    if(wv_seq[0] == 0 or wv_seq[0] == 3):
      if(a9_wv_weldingon==True):
        program_weld_on = False
        if(isHicomm):
          write_port_register(202,0)
          write_port_register(149,0)
        else:
          set_standard_digital_out(0,False)
        end
        if(wv_weldpar[2]==1):
          target_pos = feature_offset(get_actual_tcp_pose(),p[0,0,-0.01,0,0,0],wv_Line_Feature2)
          movel(target_pos,0.5,0.01)
        end
      end
    end
    background_pose = [dumy_p,dumy_p,dumy_p,dumy_p]
    move_p = background_pose
    return sin_dir
  end
  $ 151 "Reset"
  $ 152 "If Reset_Trig"
  if (Reset_Trig):
    $ 153 "Reset_Trig≔ False "
    global Reset_Trig=  False
    $ 154 "Call robotand_cell_initalizat"
    robotand_cell_initalizat()
    $ 155 "Auto_trig≔ False "
    global Auto_trig=  False
    $ 156 "write_port_register(cell_3f_2f_151,0)"
    write_port_register(cell_3f_2f_151,0)
    $ 157 "write_port_register(cell_info_152,0)"
    write_port_register(cell_info_152,0)
    $ 158 "write_port_register(weld_req_153,0)"
    write_port_register(weld_req_153,0)
    $ 159 "write_port_register(return_done_240,0)"
    write_port_register(return_done_240,0)
    $ 160 "write_port_register(robot_move_163,0)"
    write_port_register(robot_move_163,0)
    $ 161 "write_port_register(robot_pose_164,0)"
    write_port_register(robot_pose_164,0)
    $ 162 "write_port_register(182,0)"
    write_port_register(182,0)
    $ 163 "write_port_register(185,0)"
    write_port_register(185,0)
    $ 164 "write_port_register(201,0)"
    write_port_register(201,0)
    $ 165 "write_port_register(202,0)"
    write_port_register(202,0)
  end
  $ 166 "Welding_Init"
  $ 167 "'welding parameter initialization'"
  # 'welding parameter initialization'
  $ 168 "welding_etc"
  $ 196 "c5_wv_gap_y≔0"
  global c5_wv_gap_y=0
  $ 197 "c6_wv_gap_cpm≔0"
  global c6_wv_gap_cpm=0
  $ 198 "c9_wv_gap_freq≔0"
  global c9_wv_gap_freq=0
  $ 199 "c4_gap_enable≔0"
  global c4_gap_enable=0
  $ 200 "c7_wv_gap≔[c4_gap_enable,c5_wv_gap_y,c6_wv_gap_cpm,c9_wv_gap_freq]"
  global c7_wv_gap=[c4_gap_enable,c5_wv_gap_y,c6_wv_gap_cpm,c9_wv_gap_freq]
  $ 201 "init_reset_modbus_server"
  $ 202 "set_tool_voltage(24)"
  set_tool_voltage(24)
  $ 203 "write_port_register(163,0)"
  write_port_register(163,0)
  $ 204 "write_port_register(164,0)"
  write_port_register(164,0)
  $ 206 "write_port_register(201,1)"
  write_port_register(201,1)
  $ 207 "write_port_register(202,0)"
  write_port_register(202,0)
  $ 1277 "Thread_2"
  thread Thread_2():
    while (True):
      $ 1278 "Thread_heartbeat"
      $ 1279 "heartbeat≔heartbeat+1"
      global heartbeat=heartbeat+1
      $ 1280 "If heartbeat>499"
      if (heartbeat>499):
        $ 1281 "heartbeat≔0"
        global heartbeat=0
      end
      $ 1282 "write_port_register(128,heartbeat)"
      write_port_register(128,heartbeat)
      $ 1292 "Wait: 1.0"
      sleep(1.0)
    end
  end
  threadId_Thread_2 = run Thread_2()
  $ 1293 "Thread_1"
  thread Thread_1():
    while (True):
      $ 1294 "thread main"
      $ 1295 "a0_Job_Mode≔read_port_register(162)"
      global a0_Job_Mode= read_port_register (162)
      $ 1296 "a1_job_move≔read_port_register(163)"
      global a1_job_move= read_port_register (163)
      $ 1297 "If red_led≟ True "
      if (get_tool_digital_out(0) ==   True  ):
        $ 1298 "Set red_led=Off"
        set_tool_digital_out(0, False)
      end
      $ 1299 "If a0_Job_Mode≟2"
      if (a0_Job_Mode == 2):
        $ 1300 "If read_port_register(arc_onoff_168)≟2"
        if ( read_port_register (arc_onoff_168) == 2):
          $ 1301 "a9_wv_weldingon≔ True "
          global a9_wv_weldingon=  True
        else:
          $ 1302 "Else" "noBreak"
          $ 1303 "a9_wv_weldingon≔ False "
          global a9_wv_weldingon=  False
        end
        $ 1304 "If Auto_trig"
        if (Auto_trig):
          $ 1305 "get_next_number≔read_port_register(166)"
          global get_next_number= read_port_register (166)
          $ 1306 "get_move_trig≔read_port_register(167)"
          global get_move_trig= read_port_register (167)
          $ 1307 "If get_move_trig≟1 and running_trig≟ True "
          if (get_move_trig == 1  and  running_trig ==   True  ):
            $ 1308 "If get_next_number<0 or get_next_number>30"
            if (get_next_number<0  or  get_next_number>30):
              $ 1309 "write_port_register(142,141)"
              write_port_register(142,141)
              $ 1310 "Halt"
              halt
            end
            $ 1311 "If get_next_number≠Auto_cur_cell"
            if (get_next_number != Auto_cur_cell):
              $ 1312 "running_trig≔ False "
              global running_trig=  False
              $ 1313 "write_welder(0, False )"
              write_welder(0,  False  )
              $ 1314 "write_port_register(149,0)"
              write_port_register(149,0)
              $ 1315 "write_port_register(202,0)"
              write_port_register(202,0)
            else:
              $ 1316 "Else" "noBreak"
              $ 1317 "write_port_register(166,0)"
              write_port_register(166,0)
              $ 1318 "write_port_register(167,0)"
              write_port_register(167,0)
            end
          end
        end
        $ 1319 "If t_time>timer_1"
        if (t_time>timer_1):
          $ 1320 "write_port_register(143,timer_1)"
          write_port_register(143,timer_1)
        else:
          $ 1321 "Else" "noBreak"
          $ 1322 "write_port_register(143,timer_1)"
          write_port_register(143,timer_1)
          $ 1323 "write_port_register(144,timer_1)"
          write_port_register(144,timer_1)
        end
        $ 1324 "Monitoring touch and welding"
        $ 1325 "If read_welder_control(0) and read_port_register(130)≠1"
        if (read_welder_control(0)  and   read_port_register (130) != 1):
          $ 1326 "write_port_register(130,1)"
          write_port_register(130,1)
        else:
          $ 1327 "ElseIf read_welder_control(0) and read_port_register(130)≠0"
          if (read_welder_control(0)  and   read_port_register (130) != 0):
            $ 1328 "write_port_register(130,0)"
            write_port_register(130,0)
          end
        end
        $ 1329 "If read_welder(5)"
        if (read_welder(5)):
          $ 1330 "'check wcr in (digital)'"
          # 'check wcr in (digital)'
          $ 1331 "write_output_float_register(20,1)"
          write_output_float_register(20,1)
        else:
          $ 1332 "Else" "noBreak"
          $ 1333 "write_output_float_register(20,0)"
          write_output_float_register(20,0)
        end
        $ 1334 "If read_welder(4)"
        if (read_welder(4)):
          $ 1335 "'check touch (digital)'"
          # 'check touch (digital)'
          $ 1336 "write_output_float_register(21,1)"
          write_output_float_register(21,1)
        else:
          $ 1337 "Else" "noBreak"
          $ 1338 "write_output_float_register(21,0)"
          write_output_float_register(21,0)
        end
        $ 1339 "If read_welder_control(0)"
        if (read_welder_control(0)):
          $ 1340 "'check welding out (digital)'"
          # 'check welding out (digital)'
          $ 1341 "write_output_float_register(17,1)"
          write_output_float_register(17,1)
        else:
          $ 1342 "Else" "noBreak"
          $ 1343 "write_output_float_register(17,0)"
          write_output_float_register(17,0)
        end
        $ 1344 "If read_welder_control(4)"
        if (read_welder_control(4)):
          $ 1345 "'check touch out (digital)'"
          # 'check touch out (digital)'
          $ 1346 "write_output_float_register(18,1)"
          write_output_float_register(18,1)
        else:
          $ 1347 "Else" "noBreak"
          $ 1348 "write_output_float_register(18,0)"
          write_output_float_register(18,0)
        end
      end
      $ 1349 "If get_tool_digital_in(1)≟ True "
      if (get_tool_digital_in(1) ==   True  ):
        $ 1350 "set_tool_digital_out(1, False )"
        set_tool_digital_out(1,  False  )
      else:
        $ 1351 "Else" "noBreak"
        $ 1352 "set_tool_digital_out(1, True )"
        set_tool_digital_out(1,  True  )
      end
      $ 1353 "If red_led≟ True "
      if (get_tool_digital_out(0) ==   True  ):
        $ 1354 "Set red_led=Off"
        set_tool_digital_out(0, False)
        $ 1355 "end_freedrive_mode()"
        end_freedrive_mode()
      end
      $ 1356 "check_speed()"
      check_speed()
      $ 1357 "Wait: 0.05"
      sleep(0.05)
    end
  end
  threadId_Thread_1 = run Thread_1()
  thread EventThread():
    while (True):
      if (event_cal_on):
        $ 1359 "calculate_position"
        $ 1362 "move_i_f≔1"
        global move_i_f=1
        $ 1363 "get_pose_side≔0"
        global get_pose_side=0
        $ 1364 "Loop move_i_f<10"
        while (move_i_f<10):
          $ 1365 "If A_Touch_trig_l[move_i_f]≟ True "
          if (A_Touch_trig_l[move_i_f] ==   True  ):
            $ 1366 "If move_i_f≟A_VL1 or move_i_f≟A_VL2"
            if (move_i_f == A_VL1  or  move_i_f == A_VL2):
              $ 1367 "A_sel_v≔move_i_f"
              global A_sel_v=move_i_f
              $ 1368 "If simulation_mode"
              if (simulation_mode):
                $ 1369 "Call welding_parameter_sim"
                welding_parameter_sim()
              else:
                $ 1370 "Else" "noBreak"
                $ 1371 "Call welding_parameter_init"
                welding_parameter_init()
              end
              $ 1372 "If a8_wv_distance<5"
              if (a8_wv_distance<5):
                $ 1373 "write_port_register(142,143)"
                write_port_register(142,143)
                $ 1374 "Halt"
                halt
              end
              $ 1375 "b2_left_par≔ True "
              global b2_left_par=  True
              $ 1376 "b8_wv_2f≔ False "
              global b8_wv_2f=  False
              $ 1377 "If move_i_f≟A_VL2"
              if (move_i_f == A_VL2):
                $ 1378 "callar_hor≔a6_callar_hor"
                global callar_hor=a6_callar_hor
                $ 1379 "If b1_cell_info_L≟E or b1_cell_info_L≟e"
                if (b1_cell_info_L == E  or  b1_cell_info_L == e):
                  $ 1380 "'For bottom touch(zero) after offset not used now'"
                  # 'For bottom touch(zero) after offset not used now'
                  $ 1381 "vert_scallup_l≔a5_f_hole[1]"
                  global vert_scallup_l=a5_f_hole[1]
                end
                $ 1382 "b2_cell≔b1_cell_info_L"
                global b2_cell=b1_cell_info_L
              else:
                $ 1385 "Else" "noBreak"
                $ 1386 "callar_hor≔0"
                global callar_hor=0
                $ 1387 "'For bottom touch(zero) after offset not used now'"
                # 'For bottom touch(zero) after offset not used now'
                $ 1388 "vert_scallup_l≔a5_f_hole[1]"
                global vert_scallup_l=a5_f_hole[1]
                $ 1389 "b2_cell≔b1_cell_info_L"
                global b2_cell=b1_cell_info_L
              end
              $ 1390 "get_pos≔get_lr(left,a6_f_width,a5_f_hole,a7_f_distance,b2_left_par,b8_wv_2f,Touch_dis,get_margin_z,get_pose_side,callar_hor,b2_cell,center_line)"
              global get_pos=get_lr(p[.480496318984, .411279115151, .006998291210, -2.211681476386, -.899147924387, -1.383032568605],a6_f_width,a5_f_hole,a7_f_distance,b2_left_par,b8_wv_2f,Touch_dis,get_margin_z,get_pose_side,callar_hor,b2_cell,center_line)
              $ 1391 "pre_tp≔tilt_3f_fun(get_pos,[0,0,0],0)"
              global pre_tp=tilt_3f_fun(get_pos,[0,0,0],0)
              $ 1392 "A_Prepos_l[move_i_f]=pre_tp"
              A_Prepos_l[move_i_f]=pre_tp
            else:
              $ 1393 "ElseIf move_i_f≟A_VR1 or move_i_f≟A_VR2"
              if (move_i_f == A_VR1  or  move_i_f == A_VR2):
                $ 1394 "A_sel_v≔move_i_f"
                global A_sel_v=move_i_f
                $ 1395 "If simulation_mode"
                if (simulation_mode):
                  $ 1396 "Call welding_parameter_sim"
                  welding_parameter_sim()
                else:
                  $ 1397 "Else" "noBreak"
                  $ 1398 "Call welding_parameter_init"
                  welding_parameter_init()
                end
                $ 1399 "If a8_wv_distance<5"
                if (a8_wv_distance<5):
                  $ 1400 "write_port_register(142,143)"
                  write_port_register(142,143)
                  $ 1401 "Halt"
                  halt
                end
                $ 1402 "b2_left_par≔ False "
                global b2_left_par=  False
                $ 1403 "b8_wv_2f≔ False "
                global b8_wv_2f=  False
                $ 1404 "If move_i_f≟A_VR2"
                if (move_i_f == A_VR2):
                  $ 1405 "callar_hor≔a6_callar_hor"
                  global callar_hor=a6_callar_hor
                  $ 1406 "If b1_cell_info_R≟E or b1_cell_info_R≟e"
                  if (b1_cell_info_R == E  or  b1_cell_info_R == e):
                    $ 1407 "vert_scallup_r≔a5_f_hole[1]"
                    global vert_scallup_r=a5_f_hole[1]
                  end
                  $ 1408 "b2_cell≔b1_cell_info_R"
                  global b2_cell=b1_cell_info_R
                else:
                  $ 1411 "Else" "noBreak"
                  $ 1412 "callar_hor≔0"
                  global callar_hor=0
                  $ 1413 "vert_scallup_r≔a5_f_hole[1]"
                  global vert_scallup_r=a5_f_hole[1]
                  $ 1414 "b2_cell≔b1_cell_info_R"
                  global b2_cell=b1_cell_info_R
                end
                $ 1415 "get_pos≔get_lr(right,a6_f_width,a5_f_hole,a7_f_distance,b2_left_par,b8_wv_2f,Touch_dis,get_margin_z,get_pose_side,callar_hor,b2_cell,center_line)"
                global get_pos=get_lr(p[.475000000000, -.421403215678, .026417194146, 1.917761036827, -1.141682393512, 1.523356199292],a6_f_width,a5_f_hole,a7_f_distance,b2_left_par,b8_wv_2f,Touch_dis,get_margin_z,get_pose_side,callar_hor,b2_cell,center_line)
                $ 1416 "pre_tp≔tilt_3f_fun(get_pos,[0,0,0],0)"
                global pre_tp=tilt_3f_fun(get_pos,[0,0,0],0)
                $ 1417 "A_Prepos_l[move_i_f]=pre_tp"
                A_Prepos_l[move_i_f]=pre_tp
              else:
                $ 1418 "ElseIf move_i_f≟A_HOR"
                if (move_i_f == A_HOR):
                  $ 1419 "A_sel_v≔A_HOR"
                  global A_sel_v=A_HOR
                  $ 1420 "If simulation_mode"
                  if (simulation_mode):
                    $ 1421 "Call welding_parameter_sim"
                    welding_parameter_sim()
                  else:
                    $ 1422 "Else" "noBreak"
                    $ 1423 "Call welding_parameter_init"
                    welding_parameter_init()
                  end
                  $ 1424 "hor_l_scallup≔a5_f_hole[1]"
                  global hor_l_scallup=a5_f_hole[1]
                  $ 1425 "b8_wv_2f≔ True "
                  global b8_wv_2f=  True
                  $ 1426 "b2_left_par≔ True "
                  global b2_left_par=  True
                  $ 1427 "b2_cell≔b1_cell_info_L"
                  global b2_cell=b1_cell_info_L
                  $ 1428 "get_pos≔get_lr(up_left,a6_f_width,a5_f_hole,a7_f_distance,b2_left_par,b8_wv_2f,Touch_dis,get_margin_z,get_pose_side,0,b2_cell,center_line)"
                  global get_pos=get_lr(p[.492775857339, .409517380626, -.029063830209, -2.419264859926, -.998084331190, -1.368689080860],a6_f_width,a5_f_hole,a7_f_distance,b2_left_par,b8_wv_2f,Touch_dis,get_margin_z,get_pose_side,0,b2_cell,center_line)
                  $ 1429 "pre_tp≔get_pos"
                  global pre_tp=get_pos
                  $ 1430 "A_Prepos_l[move_i_f]=pre_tp"
                  A_Prepos_l[move_i_f]=pre_tp
                else:
                  $ 1431 "ElseIf move_i_f≟A_HOR_R"
                  if (move_i_f == A_HOR_R):
                    $ 1432 "A_sel_v≔A_HOR"
                    global A_sel_v=A_HOR
                    $ 1433 "If simulation_mode"
                    if (simulation_mode):
                      $ 1434 "Call welding_parameter_sim"
                      welding_parameter_sim()
                    else:
                      $ 1435 "Else" "noBreak"
                      $ 1436 "Call welding_parameter_init"
                      welding_parameter_init()
                    end
                    $ 1437 "hor_r_scallup≔a5_f_hole[2]"
                    global hor_r_scallup=a5_f_hole[2]
                    $ 1438 "b2_left_par≔ False "
                    global b2_left_par=  False
                    $ 1439 "b8_wv_2f≔ True "
                    global b8_wv_2f=  True
                    $ 1440 "b2_cell≔b1_cell_info_R"
                    global b2_cell=b1_cell_info_R
                    $ 1441 "get_pos≔get_lr(up_right,a6_f_width,a5_f_hole,a7_f_distance,b2_left_par,b8_wv_2f,Touch_dis,get_margin_z,get_pose_side,0,b2_cell,center_line)"
                    global get_pos=get_lr(p[.445203173045, -.406687378356, -.031125942276, 2.308490741423, -1.066468937023, 1.322151316133],a6_f_width,a5_f_hole,a7_f_distance,b2_left_par,b8_wv_2f,Touch_dis,get_margin_z,get_pose_side,0,b2_cell,center_line)
                    $ 1442 "pre_tp≔get_pos"
                    global pre_tp=get_pos
                    $ 1443 "A_Prepos_l[move_i_f]=pre_tp"
                    A_Prepos_l[move_i_f]=pre_tp
                  else:
                    $ 1444 "ElseIf move_i_f≟A_HOR_ML"
                    if (move_i_f == A_HOR_ML):
                      $ 1445 "A_sel_v≔A_HOR_ML"
                      global A_sel_v=A_HOR_ML
                      $ 1446 "If simulation_mode"
                      if (simulation_mode):
                        $ 1447 "Call welding_parameter_sim"
                        welding_parameter_sim()
                      else:
                        $ 1448 "Else" "noBreak"
                        $ 1449 "Call welding_parameter_init"
                        welding_parameter_init()
                      end
                      $ 1450 "b8_wv_2f≔ True "
                      global b8_wv_2f=  True
                      $ 1451 "b2_left_par≔ True "
                      global b2_left_par=  True
                      $ 1452 "b2_cell≔b1_cell_info_L"
                      global b2_cell=b1_cell_info_L
                      $ 1453 "Touch_dis≔-1*Touch_dis"
                      global Touch_dis=-1*Touch_dis
                      $ 1454 "get_pos≔get_lr(up_left,a6_f_width,a5_f_hole,a7_f_distance,b2_left_par,b8_wv_2f,Touch_dis,get_margin_z,get_pose_side,a6_callar_hor,b2_cell,center_line)"
                      global get_pos=get_lr(p[.492775857339, .409517380626, -.029063830209, -2.419264859926, -.998084331190, -1.368689080860],a6_f_width,a5_f_hole,a7_f_distance,b2_left_par,b8_wv_2f,Touch_dis,get_margin_z,get_pose_side,a6_callar_hor,b2_cell,center_line)
                      $ 1455 "Touch_dis≔-1*Touch_dis"
                      global Touch_dis=-1*Touch_dis
                      $ 1456 "pre_tp≔get_pos"
                      global pre_tp=get_pos
                      $ 1457 "A_Prepos_l[move_i_f]=pre_tp"
                      A_Prepos_l[move_i_f]=pre_tp
                    else:
                      $ 1458 "ElseIf move_i_f≟A_HOR_MR"
                      if (move_i_f == A_HOR_MR):
                        $ 1459 "A_sel_v≔A_HOR_MR"
                        global A_sel_v=A_HOR_MR
                        $ 1460 "If simulation_mode"
                        if (simulation_mode):
                          $ 1461 "Call welding_parameter_sim"
                          welding_parameter_sim()
                        else:
                          $ 1462 "Else" "noBreak"
                          $ 1463 "Call welding_parameter_init"
                          welding_parameter_init()
                        end
                        $ 1464 "b2_left_par≔ False "
                        global b2_left_par=  False
                        $ 1465 "b8_wv_2f≔ True "
                        global b8_wv_2f=  True
                        $ 1466 "b2_cell≔b1_cell_info_R"
                        global b2_cell=b1_cell_info_R
                        $ 1467 "Touch_dis≔-1*Touch_dis"
                        global Touch_dis=-1*Touch_dis
                        $ 1468 "get_pos≔get_lr(up_right,a6_f_width,a5_f_hole,a7_f_distance,b2_left_par,b8_wv_2f,Touch_dis,get_margin_z,get_pose_side,a6_callar_hor,b2_cell,center_line)"
                        global get_pos=get_lr(p[.445203173045, -.406687378356, -.031125942276, 2.308490741423, -1.066468937023, 1.322151316133],a6_f_width,a5_f_hole,a7_f_distance,b2_left_par,b8_wv_2f,Touch_dis,get_margin_z,get_pose_side,a6_callar_hor,b2_cell,center_line)
                        $ 1469 "Touch_dis≔-1*Touch_dis"
                        global Touch_dis=-1*Touch_dis
                        $ 1470 "pre_tp≔get_pos"
                        global pre_tp=get_pos
                        $ 1471 "A_Prepos_l[move_i_f]=pre_tp"
                        A_Prepos_l[move_i_f]=pre_tp
                      end
                    end
                  end
                end
              end
            end
            $ 1472 "If move_i_f≤4"
            if (move_i_f <= 4):
              $ 1473 "A_Prepos_l[move_i_f+9]=p[0,0,0,0,0,0]"
              A_Prepos_l[move_i_f+9]=p[0,0,0,0,0,0]
            end
          end
          $ 1476 "move_i_f≔move_i_f+1"
          global move_i_f=move_i_f+1
        end
        $ 1477 "event_cal_on≔ False "
        global event_cal_on=  False
      elif (event_side_on):
        $ 1479 "calculate_side"
        $ 1482 "Wait event_cal_on≟ False "
        while (not(event_cal_on ==   False  )):
          sync()
        end
        $ 1483 "move_i_f≔1"
        global move_i_f=1
        $ 1484 "get_pose_side≔get_pose_side_t"
        global get_pose_side=get_pose_side_t
        $ 1485 "Loop move_i_f<10"
        while (move_i_f<10):
          $ 1486 "If A_Touch_trig_l[move_i_f]≟ True "
          if (A_Touch_trig_l[move_i_f] ==   True  ):
            $ 1487 "If move_i_f≟A_VL1 or move_i_f≟A_VL2"
            if (move_i_f == A_VL1  or  move_i_f == A_VL2):
              $ 1488 "A_Prepos_l[move_i_f]=side_apply(A_Prepos_l[move_i_f],center_line,get_pose_side)"
              A_Prepos_l[move_i_f]=side_apply(A_Prepos_l[move_i_f],center_line,get_pose_side)
            else:
              $ 1489 "ElseIf move_i_f≟A_VR1 or move_i_f≟A_VR2"
              if (move_i_f == A_VR1  or  move_i_f == A_VR2):
                $ 1490 "A_Prepos_l[move_i_f]=side_apply(A_Prepos_l[move_i_f],center_line,get_pose_side)"
                A_Prepos_l[move_i_f]=side_apply(A_Prepos_l[move_i_f],center_line,get_pose_side)
              else:
                $ 1491 "ElseIf move_i_f≟A_HOR"
                if (move_i_f == A_HOR):
                  $ 1492 "A_Prepos_l[move_i_f]=side_apply(A_Prepos_l[move_i_f],center_line,get_pose_side)"
                  A_Prepos_l[move_i_f]=side_apply(A_Prepos_l[move_i_f],center_line,get_pose_side)
                else:
                  $ 1493 "ElseIf move_i_f≟A_HOR_R"
                  if (move_i_f == A_HOR_R):
                    $ 1494 "A_Prepos_l[move_i_f]=side_apply(A_Prepos_l[move_i_f],center_line,get_pose_side)"
                    A_Prepos_l[move_i_f]=side_apply(A_Prepos_l[move_i_f],center_line,get_pose_side)
                  else:
                    $ 1495 "ElseIf move_i_f≟A_HOR_ML"
                    if (move_i_f == A_HOR_ML):
                      $ 1496 "A_Prepos_l[move_i_f]=side_apply(A_Prepos_l[move_i_f],center_line,get_pose_side)"
                      A_Prepos_l[move_i_f]=side_apply(A_Prepos_l[move_i_f],center_line,get_pose_side)
                    else:
                      $ 1497 "ElseIf move_i_f≟A_HOR_MR"
                      if (move_i_f == A_HOR_MR):
                        $ 1498 "A_Prepos_l[move_i_f]=side_apply(A_Prepos_l[move_i_f],center_line,get_pose_side)"
                        A_Prepos_l[move_i_f]=side_apply(A_Prepos_l[move_i_f],center_line,get_pose_side)
                      end
                    end
                  end
                end
              end
            end
          end
          $ 1499 "move_i_f≔move_i_f+1"
          global move_i_f=move_i_f+1
        end
        $ 1500 "event_side_on≔ False "
        global event_side_on=  False
      elif (reset_trig):
        $ 1502 "Call reset_weld_param"
        reset_weld_param()
        $ 1503 "reset_trig≔ False "
        global reset_trig=  False
      elif (time_cal_trig):
        $ 1505 "t_time≔time_cal(Auto_W_num,Auto_total_cell,A_Speed_list,A_Distance_list,A_Touch_p,0)"
        global t_time=time_cal(Auto_W_num,Auto_total_cell,A_Speed_list,A_Distance_list,A_Touch_p,0)
        $ 1506 "write_port_register(144,t_time)"
        write_port_register(144,t_time)
        $ 1507 "time_cal_trig≔ False "
        global time_cal_trig=  False
      elif (pause_trig):
        $ 1509 "s_conn≔socket_open('192.168.1.7',29999)"
        global s_conn=socket_open("192.168.1.7",29999)
        $ 1510 "s_send≔socket_send_string('pause')"
        global s_send=socket_send_string("pause")
        $ 1511 "s_send≔socket_send_byte(10)"
        global s_send=socket_send_byte(10)
        $ 1512 "socket_close()"
        socket_close()
        $ 1513 "pause_trig≔ False "
        global pause_trig=  False
      end
      sync()
    end
  end
  eventThread = run EventThread()
  while (True):
    $ 208 "Robot Program"
    $ 226 "If simulation_mode"
    if (simulation_mode):
      $ 227 "'work mode 2'"
      # 'work mode 2'
      $ 228 "write_port_register(162,2)"
      write_port_register(162,2)
      $ 229 "touch_temp≔0"
      global touch_temp=0
    end
    $ 230 "If a0_Job_Mode≟1"
    if (a0_Job_Mode == 1):
      $ 231 "job mode 1"
      $ 232 "'JOB_MANUAL'"
      # 'JOB_MANUAL'
      $ 233 "write_port_register(robot_ready_141,1)"
      write_port_register(robot_ready_141,1)
      $ 234 "If freedrive≟ True  and freedrive_trg≟ False "
      if (get_tool_digital_in(1) ==   True    and  freedrive_trg ==   False  ):
        $ 235 "freedrive_trg≔ True "
        global freedrive_trg=  True
        $ 236 "freedrive_mode()"
        freedrive_mode()
      else:
        $ 237 "ElseIf freedrive≟ False  and freedrive_trg≟ True "
        if (get_tool_digital_in(1) ==   False    and  freedrive_trg ==   True  ):
          $ 238 "end_freedrive_mode()"
          end_freedrive_mode()
          $ 239 "freedrive_trg≔ False "
          global freedrive_trg=  False
        end
      end
      $ 243 "If freedrive≟ True  and save_tool≟ True "
      if (get_tool_digital_in(1) ==   True    and  get_tool_digital_in(0) ==   True  ):
        $ 247 "Wait: 0.01"
        sleep(0.01)
      else:
        $ 248 "ElseIf a1_job_move≟1"
        if (a1_job_move == 1):
          $ 249 "'Manual - Move Home/Packing/Warmup'"
          # 'Manual - Move Home/Packing/Warmup'
          $ 250 "If read_port_register(robot_pose_164)≟1"
          if ( read_port_register (robot_pose_164) == 1):
            $ 251 "write_port_register(robot_ready_141,0)"
            write_port_register(robot_ready_141,0)
            $ 252 "homeing()"
            homeing()
            $ 253 "MoveJ"
            $ 254 "Packing_pos" "breakAfter"
            movej([1.5877798795700073, -0.0173419157611292, -2.4983108679400843, -1.4065726439105433, 1.626846194267273, 3.0169763565063477], a=0.9599310885968813, v=0.9599310885968813)
          else:
            $ 255 "ElseIf read_port_register(robot_pose_164)≟2"
            if ( read_port_register (robot_pose_164) == 2):
              $ 256 "write_port_register(robot_ready_141,0)"
              write_port_register(robot_ready_141,0)
              $ 257 "homeing()"
              homeing()
            else:
              $ 258 "ElseIf read_port_register(robot_pose_164)≟3"
              global thread_flag_258=0
              thread Thread_if_258():
                $ 259 "write_port_register(robot_ready_141,0)"
                write_port_register(robot_ready_141,0)
                $ 260 "Warm-up"
                $ 261 "Loop 22 times"
                Loop_9 = 0
                while (Loop_9 < 22):
                  $ 262 "MoveJ"
                  $ 263 "Warming_1" "breakAfter"
                  movej([1.0598392486572266, -1.0896032492267054, -1.2158034483539026, -2.3403762022601526, 1.497584342956543, 2.354665517807007], a=0.17453292519943295, v=0.08726646259971647)
                  $ 264 "Warming_2" "breakAfter"
                  movej([0.7106529474258423, -1.0894954840289515, -1.215731445943014, -2.3402441183673304, 1.4977161884307861, 2.3545455932617188], a=0.17453292519943295, v=0.08726646259971647)
                  $ 265 "Warming_3" "breakAfter"
                  movej([0.8852421641349792, -1.0894234816180628, -1.215863052998678, -2.340435806904928, 1.497644305229187, 2.3545212745666504], a=0.17453292519943295, v=0.08726646259971647)
                  $ 266 "Warming_4" "breakAfter"
                  movej([0.885266125202179, -1.263935391102926, -1.2099388281451624, -2.352635685597555, 1.4888625144958496, 2.3787333965301514], a=0.17453292519943295, v=0.08726646259971647)
                  $ 267 "Wariming_5" "breakAfter"
                  movej([0.8852541446685791, -0.9149578253375452, -1.217938248311178, -2.335618321095602, 1.501125693321228, 2.3452301025390625], a=0.17453292519943295, v=0.08726646259971647)
                  $ 268 "Warming_6" "breakAfter"
                  movej([0.8852177858352661, -1.0895074049579065, -1.3828147093402308, -2.343850914631979, 1.489568829536438, 2.3598153591156006], a=0.17453292519943295, v=0.08726646259971647)
                  $ 269 "Warming_7" "breakAfter"
                  movej([0.885229766368866, -1.0894115606891077, -1.220372502003805, -2.335630242024557, 1.5009583234786987, 2.3453502655029297], a=0.17453292519943295, v=0.08726646259971647)
                  $ 270 "Warming_8" "breakAfter"
                  movej([0.6920775233962951, -1.0506328608604214, -1.2152130579572011, -2.5072867131215766, 1.4917910996963177, 2.3459413556024855], a=0.17453292519943295, v=0.08726646259971647)
                  $ 271 "Warming_9" "breakAfter"
                  movej([0.6929177641868591, -1.0475013891803187, -1.2503178755389612, -2.327541176472799, 1.5014369487762451, 2.345398187637329], a=0.17453292519943295, v=0.08726646259971647)
                  $ 272 "Warming_10" "breakAfter"
                  movej([0.8162043690681458, -1.1462538878070276, -1.3285825888263147, -2.3897975126849573, 1.2906681299209595, 2.3704988956451416], a=0.17453292519943295, v=0.08726646259971647)
                  $ 273 "Warming_11" "breakAfter"
                  movej([0.6952417412291937, -1.0226626805382075, -1.3187663864026051, -2.3852732107244847, 1.5281305955128988, 2.3484138521676003], a=0.17453292519943295, v=0.08726646259971647)
                  $ 274 "Warming_12" "breakAfter"
                  movej([0.6938896179199219, -1.0222962538348597, -1.3204510847674769, -2.403698269520895, 1.7271294593811035, 2.3448219299316406], a=0.17453292519943295, v=0.08726646259971647)
                  $ 275 "Warming_13" "breakAfter"
                  movej([0.685538113117218, -1.038980786000387, -1.3163254896747034, -2.3712590376483362, 1.5282130241394043, 2.0345256328582764], a=0.17453292519943295, v=0.08726646259971647)
                  $ 276 "Warming_14" "breakAfter"
                  movej([0.721284806728363, -1.0075753370868128, -1.3205111662494105, -2.399587933217184, 1.5282011032104492, 2.539506673812866], a=0.17453292519943295, v=0.08726646259971647)
                  Loop_9 = Loop_9 + 1
                end
                $ 277 "homeing()"
                homeing()
                $ 278 "Wait: 2.0"
                sleep(2.0)
                thread_flag_258 = 1
              end
              if ( read_port_register (robot_pose_164) == 3):
                global thread_handler_258=run Thread_if_258()
                while (thread_flag_258 == 0):
                  if not( read_port_register (robot_pose_164) == 3):
                    kill thread_handler_258
                    thread_flag_258 = 2
                  else:
                    sync()
                  end
                end
              else:
                thread_flag_258 = 2
              end
              if (thread_flag_258 == 2):
                $ 279 "ElseIf read_port_register(robot_pose_164)≟4"
                if ( read_port_register (robot_pose_164) == 4):
                  $ 280 "write_port_register(robot_ready_141,0)"
                  write_port_register(robot_ready_141,0)
                  $ 281 "homeing()"
                  homeing()
                  $ 282 "MoveJ"
                  $ 283 "pre_mounting" "breakAfter"
                  movej([1.2356762886047363, -0.8703244368182581, -0.942230526600973, -2.3905327955829065, 1.3216267824172974, 2.6514604091644287], a=0.7853981633974483, v=0.7853981633974483)
                  $ 284 "Mounting_pos" "breakAfter"
                  movej([0.6231353085164267, -0.6300961531972575, -0.9034285948871803, -1.770059340221131, 1.417516049558281, 1.7792033261567348], a=0.7853981633974483, v=0.7853981633974483)
                else:
                  $ 285 "ElseIf read_port_register(robot_pose_164)≟5"
                  if ( read_port_register (robot_pose_164) == 5):
                    $ 286 "c_p≔get_actual_tcp_pose()"
                    global c_p= get_actual_tcp_pose ()
                    $ 287 "MoveL"
                    $ 288 "m_p≔pose_trans(c_p, p[0,0,0,d2r(tilt_deg_man),0,0])"
                    global m_p= pose_trans (c_p, p[0,0,0,d2r(tilt_deg_man),0,0])
                    $ 289 "m_p" "breakAfter"
                    movel(pose_trans(Base, m_p), a=0.03, v=0.03)
                    $ 290 "m_p≔pose_trans(c_p, p[0,0,0,d2r(-tilt_deg_man),0,0])"
                    global m_p= pose_trans (c_p, p[0,0,0,d2r(-tilt_deg_man),0,0])
                    $ 291 "m_p" "breakAfter"
                    movel(pose_trans(Base, m_p), a=0.03, v=0.03)
                    $ 292 "c_p" "breakAfter"
                    movel(pose_trans(Base, c_p), a=0.03, v=0.03)
                    $ 293 "m_p≔pose_trans(c_p, p[0,0,0,0,d2r(tilt_deg_man),0])"
                    global m_p= pose_trans (c_p, p[0,0,0,0,d2r(tilt_deg_man),0])
                    $ 294 "m_p" "breakAfter"
                    movel(pose_trans(Base, m_p), a=0.03, v=0.03)
                    $ 295 "m_p≔pose_trans(c_p, p[0,0,0,0,d2r(-tilt_deg_man),0])"
                    global m_p= pose_trans (c_p, p[0,0,0,0,d2r(-tilt_deg_man),0])
                    $ 296 "m_p" "breakAfter"
                    movel(pose_trans(Base, m_p), a=0.03, v=0.03)
                    $ 297 "c_p" "breakAfter"
                    movel(pose_trans(Base, c_p), a=0.03, v=0.03)
                    $ 298 "m_p≔pose_trans(c_p, p[0,0,0,0,0,d2r(tilt_deg_man)])"
                    global m_p= pose_trans (c_p, p[0,0,0,0,0,d2r(tilt_deg_man)])
                    $ 299 "m_p" "breakAfter"
                    movel(pose_trans(Base, m_p), a=0.03, v=0.03)
                    $ 300 "m_p≔pose_trans(c_p, p[0,0,0,0,0,d2r(-tilt_deg_man)])"
                    global m_p= pose_trans (c_p, p[0,0,0,0,0,d2r(-tilt_deg_man)])
                    $ 301 "m_p" "breakAfter"
                    movel(pose_trans(Base, m_p), a=0.03, v=0.03)
                    $ 302 "c_p" "breakAfter"
                    movel(pose_trans(Base, c_p), a=0.03, v=0.03)
                  end
                end
              end
            end
          end
          $ 303 "Call Move_done"
          Move_done()
        end
      end
      $ 304 "Call robotand_cell_initalizat"
      robotand_cell_initalizat()
    else:
      $ 305 "ElseIf a0_Job_Mode≟2"
      global thread_flag_305=0
      thread Thread_if_305():
        $ 306 "'JOB_AUTO'"
        # 'JOB_AUTO'
        $ 307 "auto_on≔ True "
        global auto_on=  True
        $ 308 "Init"
        $ 309 "If freedrive_trg"
        if (freedrive_trg):
          $ 310 "end_freedrive_mode()"
          end_freedrive_mode()
          $ 311 "freedrive_trg≔ False "
          global freedrive_trg=  False
        end
        $ 312 "write_port_register(202,0)"
        write_port_register(202,0)
        $ 313 "write_port_register(robot_ready_141,0)"
        write_port_register(robot_ready_141,0)
        $ 314 "homeing()"
        homeing()
        $ 315 "Wait: 0.2"
        sleep(0.2)
        $ 316 "Cell_calculation"
        $ 317 "'setting'"
        # 'setting'
        $ 318 "Auto_trig≔ False "
        global Auto_trig=  False
        $ 319 "If Auto_trig≟ False "
        if (Auto_trig ==   False  ):
          $ 320 "If simulation_mode"
          if (simulation_mode):
            $ 321 "b1_cell_info_L≔B"
            global b1_cell_info_L=B
            $ 322 "b1_cell_info_R≔B"
            global b1_cell_info_R=B
            $ 323 "b1_cell_select≔motion_num([A_VL1,A_VR1,A_HOR,0,0,0])"
            global b1_cell_select=motion_num([A_VL1,A_VR1,A_HOR,0,0,0])
            $ 324 "b1_cell_select≔motion_num([A_HOR,0,0,0,0,0])"
            global b1_cell_select=motion_num([A_HOR,0,0,0,0,0])
            $ 325 "EXT_flag1≔integer_to_binary_list(read_port_register(2048))"
            global EXT_flag1= integer_to_binary_list ( read_port_register (2048))
            $ 326 "b1_cell_thickne≔6"
            global b1_cell_thickne=6
            $ 327 "A_Touch_trig_l≔touch_cal(b1_cell_info_L,b1_cell_info_R,b1_cell_select)"
            global A_Touch_trig_l=touch_cal(b1_cell_info_L,b1_cell_info_R,b1_cell_select)
            $ 328 "Auto_W_num≔cell_motion(A_Touch_trig_l,b1_cell_thickne,EXT_flag1,b1_cell_info_L,b1_cell_info_R)"
            global Auto_W_num=cell_motion(A_Touch_trig_l,b1_cell_thickne,EXT_flag1,b1_cell_info_L,b1_cell_info_R)
            $ 330 "Auto_total_cell≔cell_num(Auto_W_num)"
            global Auto_total_cell=cell_num(Auto_W_num)
            $ 331 "Auto_trig≔ True "
            global Auto_trig=  True
            $ 332 "A_sel_v≔Auto_W_num[0]"
            global A_sel_v=Auto_W_num[0]
          else:
            $ 333 "Else" "noBreak"
            $ 334 "b1_cell_info_L≔read_port_register(171)"
            global b1_cell_info_L= read_port_register (171)
            $ 335 "b1_cell_info_R≔read_port_register(172)"
            global b1_cell_info_R= read_port_register (172)
            $ 336 "EXT_flag1≔integer_to_binary_list(read_port_register(179))"
            global EXT_flag1= integer_to_binary_list ( read_port_register (179))
            $ 337 "b1_cell_select≔read_port_register(178)"
            global b1_cell_select= read_port_register (178)
            $ 338 "b1_cell_thickne≔read_port_register(183)"
            global b1_cell_thickne= read_port_register (183)
            $ 339 "A_Touch_trig_l≔touch_cal(b1_cell_info_L,b1_cell_info_R,b1_cell_select)"
            global A_Touch_trig_l=touch_cal(b1_cell_info_L,b1_cell_info_R,b1_cell_select)
            $ 340 "Auto_W_num≔cell_motion(A_Touch_trig_l,b1_cell_thickne,EXT_flag1,b1_cell_info_L,b1_cell_info_R)"
            global Auto_W_num=cell_motion(A_Touch_trig_l,b1_cell_thickne,EXT_flag1,b1_cell_info_L,b1_cell_info_R)
            $ 341 "Auto_total_cell≔cell_num(Auto_W_num)"
            global Auto_total_cell=cell_num(Auto_W_num)
            $ 342 "Auto_trig≔ True "
            global Auto_trig=  True
            $ 343 "A_sel_v≔Auto_W_num[0]"
            global A_sel_v=Auto_W_num[0]
          end
          $ 344 "write_port_register(139,Auto_total_cell-1)"
          write_port_register(139,Auto_total_cell-1)
        end
        $ 345 "Auto_cur_cell≔0"
        global Auto_cur_cell=0
        $ 346 "Touch,Welding"
        $ 347 "'Calculate total sequence and decide way'"
        # 'Calculate total sequence and decide way'
        $ 348 "Calculate & Move & Touch"
        $ 349 "touch_init"
        $ 350 "Call cell_info"
        cell_info()
        $ 351 "If simulation_mode"
        if (simulation_mode):
          $ 352 "Call welding_parameter_sim"
          welding_parameter_sim()
        else:
          $ 353 "Else" "noBreak"
          $ 354 "Call welding_parameter_init"
          welding_parameter_init()
          $ 355 "touch_temp≔read_port_register(180)"
          global touch_temp= read_port_register (180)
          $ 356 "A_cur_2f≔0"
          global A_cur_2f=0
          $ 357 "wv_direction≔1"
          global wv_direction=1
        end
        $ 358 "If touch_temp≟0"
        if (touch_temp == 0):
          $ 359 "reset Variable"
          $ 360 "A_Prepos_l=[p[0, 0, 0, 0, 0, 0], p[0, 0, 0, 0, 0, 0], p[0, 0, 0, 0, 0, 0],p[0, 0, 0, 0, 0, 0], p[0, 0, 0, 0, 0, 0], p[0, 0, 0, 0, 0, 0], p[0, 0, 0, 0, 0, 0], p[0, 0, 0, 0, 0, 0], p[0, 0, 0, 0, 0, 0], p[0, 0, 0, 0, 0, 0], p[0, 0, 0, 0, 0, 0],p[0, 0, 0, 0, 0, 0],p[0, 0, 0, 0, 0, 0],p[0, 0, 0, 0, 0, 0],p[0, 0, 0, 0, 0, 0],p[0,0,0,0,0,0]]"
          A_Prepos_l=[p[0, 0, 0, 0, 0, 0], p[0, 0, 0, 0, 0, 0], p[0, 0, 0, 0, 0, 0],p[0, 0, 0, 0, 0, 0], p[0, 0, 0, 0, 0, 0], p[0, 0, 0, 0, 0, 0], p[0, 0, 0, 0, 0, 0], p[0, 0, 0, 0, 0, 0], p[0, 0, 0, 0, 0, 0], p[0, 0, 0, 0, 0, 0], p[0, 0, 0, 0, 0, 0],p[0, 0, 0, 0, 0, 0],p[0, 0, 0, 0, 0, 0],p[0, 0, 0, 0, 0, 0],p[0, 0, 0, 0, 0, 0],p[0,0,0,0,0,0]]
          $ 361 "A_Touch_p=[p[0, 0, 0, 0, 0, 0], p[0, 0, 0, 0, 0, 0], p[0, 0, 0, 0, 0, 0],p[0, 0, 0, 0, 0, 0], p[0, 0, 0, 0, 0, 0], p[0, 0, 0, 0, 0, 0], p[0, 0, 0, 0, 0, 0], p[0, 0, 0, 0, 0, 0], p[0, 0, 0, 0, 0, 0], p[0, 0, 0, 0, 0, 0], p[0, 0, 0, 0, 0, 0],p[0, 0, 0, 0, 0, 0],p[0, 0, 0, 0, 0, 0],p[0, 0, 0, 0, 0, 0],p[0, 0, 0, 0, 0, 0],p[0,0,0,0,0,0]]"
          A_Touch_p=[p[0, 0, 0, 0, 0, 0], p[0, 0, 0, 0, 0, 0], p[0, 0, 0, 0, 0, 0],p[0, 0, 0, 0, 0, 0], p[0, 0, 0, 0, 0, 0], p[0, 0, 0, 0, 0, 0], p[0, 0, 0, 0, 0, 0], p[0, 0, 0, 0, 0, 0], p[0, 0, 0, 0, 0, 0], p[0, 0, 0, 0, 0, 0], p[0, 0, 0, 0, 0, 0],p[0, 0, 0, 0, 0, 0],p[0, 0, 0, 0, 0, 0],p[0, 0, 0, 0, 0, 0],p[0, 0, 0, 0, 0, 0],p[0,0,0,0,0,0]]
          $ 362 "reset_par"
          $ 363 "for_cal_rot≔p[0,0,0,0,0,0]"
          global for_cal_rot=p[0,0,0,0,0,0]
          $ 364 "for_cal_zr≔p[0,0,0,0,0,0]"
          global for_cal_zr=p[0,0,0,0,0,0]
          $ 365 "for_z_VLR2≔p[0,0,0,0,0,0]"
          global for_z_VLR2=p[0,0,0,0,0,0]
          $ 366 "for_cal_x_wel≔p[0,0,0,0,0,0]"
          global for_cal_x_wel=p[0,0,0,0,0,0]
          $ 367 "for_cal_xy≔p[0,0,0,0,0,0]"
          global for_cal_xy=p[0,0,0,0,0,0]
          $ 368 "for_cal_y_wel≔p[0,0,0,0,0,0]"
          global for_cal_y_wel=p[0,0,0,0,0,0]
          $ 369 "for_x_HOR≔p[0,0,0,0,0,0]"
          global for_x_HOR=p[0,0,0,0,0,0]
          $ 370 "for_x_HOR_R≔p[0,0,0,0,0,0]"
          global for_x_HOR_R=p[0,0,0,0,0,0]
          $ 371 "for_z_VL1≔p[0,0,0,0,0,0]"
          global for_z_VL1=p[0,0,0,0,0,0]
          $ 372 "for_z_VR1≔p[0,0,0,0,0,0]"
          global for_z_VR1=p[0,0,0,0,0,0]
        end
        $ 373 "write_port_register(143,0)"
        write_port_register(143,0)
        $ 374 "write_port_register(144,0)"
        write_port_register(144,0)
        $ 375 "timer_1: Reset"
        timer_1 = 0
        $ 376 "EXT_flag1≔integer_to_binary_list(read_port_register(179))"
        global EXT_flag1= integer_to_binary_list ( read_port_register (179))
        $ 378 "If touch_temp≟0"
        if (touch_temp == 0):
          $ 379 "write_port_register(138,0)"
          write_port_register(138,0)
          $ 380 "get_touch_position"
          $ 381 "get pre-positions"
          $ 382 "If read_port_register(work_type_165)≟2"
          if ( read_port_register (work_type_165) == 2):
            $ 383 "freedrive touch"
            $ 384 "move_i≔1"
            global move_i=1
            $ 385 "Loop move_i<9"
            while (move_i<9):
              $ 386 "Wait: 0.1"
              sleep(0.1)
              $ 387 "Wait save_tool=LO"
              while (get_tool_digital_in(0) == True):
                sync()
              end
              $ 388 "If A_Touch_trig_l[move_i]≟ True "
              if (A_Touch_trig_l[move_i] ==   True  ):
                $ 389 "If move_i≟A_HOR"
                if (move_i == A_HOR):
                  $ 390 "If b1_cell_info_L≟B or b1_cell_info_L≟D or b1_cell_info_L≟d or A_Prepos_l[A_VL1]≟p[0,0,0,0,0,0]"
                  if (b1_cell_info_L == B  or  b1_cell_info_L == D  or  b1_cell_info_L == d  or  A_Prepos_l[A_VL1] == p[0,0,0,0,0,0]):
                    $ 391 "write_port_register(touch_cell_155,5)"
                    write_port_register(touch_cell_155,5)
                    $ 392 "write_port_register(touch_num_156,1)"
                    write_port_register(touch_num_156,1)
                    $ 393 "Call touch_sub"
                    touch_sub()
                    $ 394 "g_cp≔get_actual_tcp_pose()"
                    global g_cp= get_actual_tcp_pose ()
                    $ 395 "If g_cp[2]<(get_margin_z+a7_cell_bottom)/1000"
                    if (g_cp[2]<(get_margin_z+a7_cell_bottom)/1000):
                      $ 396 "g_cp[2]=(get_margin_z+a7_cell_bottom)/1000"
                      g_cp[2]=(get_margin_z+a7_cell_bottom)/1000
                    end
                    $ 397 "A_Prepos_l[move_i]=g_cp"
                    A_Prepos_l[move_i]=g_cp
                  end
                else:
                  $ 398 "ElseIf move_i≟A_HOR_ML"
                  if (move_i == A_HOR_ML):
                    $ 399 "If b1_cell_info_L≟B or b1_cell_info_L≟D or b1_cell_info_L≟d or A_Prepos_l[A_VL1]≟p[0,0,0,0,0,0]"
                    if (b1_cell_info_L == B  or  b1_cell_info_L == D  or  b1_cell_info_L == d  or  A_Prepos_l[A_VL1] == p[0,0,0,0,0,0]):
                      $ 400 "write_port_register(touch_cell_155,5)"
                      write_port_register(touch_cell_155,5)
                      $ 401 "write_port_register(touch_num_156,3)"
                      write_port_register(touch_num_156,3)
                      $ 402 "Call touch_sub"
                      touch_sub()
                      $ 403 "g_cp≔get_actual_tcp_pose()"
                      global g_cp= get_actual_tcp_pose ()
                      $ 404 "If g_cp[2]<(get_margin_z+a7_cell_bottom)/1000"
                      if (g_cp[2]<(get_margin_z+a7_cell_bottom)/1000):
                        $ 405 "g_cp[2]=(get_margin_z+a7_cell_bottom)/1000"
                        g_cp[2]=(get_margin_z+a7_cell_bottom)/1000
                      end
                      $ 406 "A_Prepos_l[move_i]=g_cp"
                      A_Prepos_l[move_i]=g_cp
                    end
                  else:
                    $ 407 "ElseIf move_i≟A_HOR_R"
                    if (move_i == A_HOR_R):
                      $ 408 "If b1_cell_info_L≟B or b1_cell_info_L≟D or b1_cell_info_L≟d or A_Prepos_l[A_VL1]≟p[0,0,0,0,0,0]"
                      if (b1_cell_info_L == B  or  b1_cell_info_L == D  or  b1_cell_info_L == d  or  A_Prepos_l[A_VL1] == p[0,0,0,0,0,0]):
                        $ 409 "write_port_register(touch_cell_155,5)"
                        write_port_register(touch_cell_155,5)
                        $ 410 "write_port_register(touch_num_156,2)"
                        write_port_register(touch_num_156,2)
                        $ 411 "Call touch_sub"
                        touch_sub()
                        $ 412 "g_cp≔get_actual_tcp_pose()"
                        global g_cp= get_actual_tcp_pose ()
                        $ 413 "If g_cp[2]<(get_margin_z+a7_cell_bottom)/1000"
                        if (g_cp[2]<(get_margin_z+a7_cell_bottom)/1000):
                          $ 414 "g_cp[2]=(get_margin_z+a7_cell_bottom)/1000"
                          g_cp[2]=(get_margin_z+a7_cell_bottom)/1000
                        end
                        $ 415 "A_Prepos_l[move_i]=g_cp"
                        A_Prepos_l[move_i]=g_cp
                      end
                    else:
                      $ 416 "ElseIf move_i≟A_HOR_MR"
                      if (move_i == A_HOR_MR):
                        $ 417 "If b1_cell_info_L≟B or b1_cell_info_L≟D or b1_cell_info_L≟d or A_Prepos_l[A_VL1]≟p[0,0,0,0,0,0]"
                        if (b1_cell_info_L == B  or  b1_cell_info_L == D  or  b1_cell_info_L == d  or  A_Prepos_l[A_VL1] == p[0,0,0,0,0,0]):
                          $ 418 "write_port_register(touch_cell_155,5)"
                          write_port_register(touch_cell_155,5)
                          $ 419 "write_port_register(touch_num_156,4)"
                          write_port_register(touch_num_156,4)
                          $ 420 "Call touch_sub"
                          touch_sub()
                          $ 421 "g_cp≔get_actual_tcp_pose()"
                          global g_cp= get_actual_tcp_pose ()
                          $ 422 "If g_cp[2]<(get_margin_z+a7_cell_bottom)/1000"
                          if (g_cp[2]<(get_margin_z+a7_cell_bottom)/1000):
                            $ 423 "g_cp[2]=(get_margin_z+a7_cell_bottom)/1000"
                            g_cp[2]=(get_margin_z+a7_cell_bottom)/1000
                          end
                          $ 424 "A_Prepos_l[move_i]=g_cp"
                          A_Prepos_l[move_i]=g_cp
                        end
                      else:
                        $ 425 "Else" "noBreak"
                        $ 426 "write_port_register(touch_cell_155,move_i)"
                        write_port_register(touch_cell_155,move_i)
                        $ 427 "write_port_register(touch_num_156,1)"
                        write_port_register(touch_num_156,1)
                        $ 428 "Call touch_sub"
                        touch_sub()
                        $ 429 "A_Prepos_l[move_i]=get_actual_tcp_pose()"
                        A_Prepos_l[move_i]= get_actual_tcp_pose ()
                        $ 430 "If move_i≤4"
                        if (move_i <= 4):
                          $ 431 "write_port_register(touch_cell_155,move_i)"
                          write_port_register(touch_cell_155,move_i)
                          $ 432 "write_port_register(touch_num_156,2)"
                          write_port_register(touch_num_156,2)
                          $ 433 "Wait: 0.1"
                          sleep(0.1)
                          $ 434 "Call touch_sub"
                          touch_sub()
                          $ 435 "A_Prepos_l[move_i+9]=get_actual_tcp_pose()"
                          A_Prepos_l[move_i+9]= get_actual_tcp_pose ()
                        end
                      end
                    end
                  end
                end
              else:
                $ 436 "Else" "noBreak"
                $ 437 "A_Prepos_l[move_i]=p[0,0,0,0,0,0]"
                A_Prepos_l[move_i]=p[0,0,0,0,0,0]
                $ 438 "If move_i≤4"
                if (move_i <= 4):
                  $ 439 "A_Prepos_l[move_i+7]=p[0,0,0,0,0,0]"
                  A_Prepos_l[move_i+7]=p[0,0,0,0,0,0]
                else:
                  $ 440 "ElseIf move_i≟A_HOR"
                  if (move_i == A_HOR):
                    $ 441 "A_Prepos_l[A_HOR_ML]=p[0,0,0,0,0,0]"
                    A_Prepos_l[A_HOR_ML]=p[0,0,0,0,0,0]
                    $ 442 "A_Prepos_l[A_HOR_MR]=p[0,0,0,0,0,0]"
                    A_Prepos_l[A_HOR_MR]=p[0,0,0,0,0,0]
                    $ 443 "A_Prepos_l[A_HOR_M]=p[0,0,0,0,0,0]"
                    A_Prepos_l[A_HOR_M]=p[0,0,0,0,0,0]
                    $ 444 "A_Prepos_l[A_HOR_R]=p[0,0,0,0,0,0]"
                    A_Prepos_l[A_HOR_R]=p[0,0,0,0,0,0]
                  end
                end
              end
              $ 445 "move_i≔move_i+1"
              global move_i=move_i+1
            end
            $ 446 "change deg"
            $ 447 "move_i≔1"
            global move_i=1
            $ 448 "Loop move_i<14"
            while (move_i<14):
              $ 449 "If A_Prepos_l[move_i]≠p[0,0,0,0,0,0]"
              if (A_Prepos_l[move_i] != p[0,0,0,0,0,0]):
                $ 450 "If move_i≟A_VL1 or move_i≟A_VL2 or move_i≟A_VL1_END or move_i≟A_VL2_END"
                if (move_i == A_VL1  or  move_i == A_VL2  or  move_i == A_VL1_END  or  move_i == A_VL2_END):
                  $ 451 "b2_left_par≔ True "
                  global b2_left_par=  True
                  $ 452 "b8_wv_2f≔ False "
                  global b8_wv_2f=  False
                  $ 453 "get_pos≔A_Prepos_l[move_i]"
                  global get_pos=A_Prepos_l[move_i]
                  $ 454 "get_org≔left"
                  global get_org=p[.480496318984, .411279115151, .006998291210, -2.211681476386, -.899147924387, -1.383032568605]
                  $ 455 "get_pos≔p[get_pos[0],get_pos[1],get_pos[2],get_org[3],get_org[4],get_org[5]]"
                  global get_pos=p[get_pos[0],get_pos[1],get_pos[2],get_org[3],get_org[4],get_org[5]]
                  $ 456 "pre_tp≔tilt_3f_fun(get_pos,[0,0],a5_f_hole[1])"
                  global pre_tp=tilt_3f_fun(get_pos,[0,0],a5_f_hole[1])
                else:
                  $ 457 "ElseIf move_i≟A_VR1 or move_i≟A_VR2 or move_i≟A_VR1_END or move_i≟A_VR2_END"
                  if (move_i == A_VR1  or  move_i == A_VR2  or  move_i == A_VR1_END  or  move_i == A_VR2_END):
                    $ 458 "b2_left_par≔ False "
                    global b2_left_par=  False
                    $ 459 "b8_wv_2f≔ False "
                    global b8_wv_2f=  False
                    $ 460 "get_pos≔A_Prepos_l[move_i]"
                    global get_pos=A_Prepos_l[move_i]
                    $ 461 "get_org≔right"
                    global get_org=p[.475000000000, -.421403215678, .026417194146, 1.917761036827, -1.141682393512, 1.523356199292]
                    $ 462 "get_pos≔p[get_pos[0],get_pos[1],get_pos[2],get_org[3],get_org[4],get_org[5]]"
                    global get_pos=p[get_pos[0],get_pos[1],get_pos[2],get_org[3],get_org[4],get_org[5]]
                    $ 463 "pre_tp≔tilt_3f_fun(get_pos,[0,0],a5_f_hole[1])"
                    global pre_tp=tilt_3f_fun(get_pos,[0,0],a5_f_hole[1])
                  else:
                    $ 464 "ElseIf move_i≟A_HOR or move_i≟A_HOR_ML"
                    if (move_i == A_HOR  or  move_i == A_HOR_ML):
                      $ 465 "b8_wv_2f≔ True "
                      global b8_wv_2f=  True
                      $ 466 "b2_left_par≔ True "
                      global b2_left_par=  True
                      $ 467 "get_pos≔A_Prepos_l[move_i]"
                      global get_pos=A_Prepos_l[move_i]
                      $ 468 "get_org≔up_left"
                      global get_org=p[.492775857339, .409517380626, -.029063830209, -2.419264859926, -.998084331190, -1.368689080860]
                      $ 469 "get_pos≔p[get_pos[0],get_pos[1],get_pos[2],get_org[3],get_org[4],get_org[5]]"
                      global get_pos=p[get_pos[0],get_pos[1],get_pos[2],get_org[3],get_org[4],get_org[5]]
                      $ 470 "pre_tp≔tilt_2f_fun(get_pos,[0,0], True , True )"
                      global pre_tp=tilt_2f_fun(get_pos,[0,0],  True  ,  True  )
                    else:
                      $ 471 "ElseIf move_i≟A_HOR_R or move_i≟A_HOR_MR"
                      if (move_i == A_HOR_R  or  move_i == A_HOR_MR):
                        $ 472 "b8_wv_2f≔ True "
                        global b8_wv_2f=  True
                        $ 473 "b2_left_par≔ False "
                        global b2_left_par=  False
                        $ 474 "get_pos≔A_Prepos_l[move_i]"
                        global get_pos=A_Prepos_l[move_i]
                        $ 475 "get_org≔up_right"
                        global get_org=p[.445203173045, -.406687378356, -.031125942276, 2.308490741423, -1.066468937023, 1.322151316133]
                        $ 476 "get_pos≔p[get_pos[0],get_pos[1],get_pos[2],get_org[3],get_org[4],get_org[5]]"
                        global get_pos=p[get_pos[0],get_pos[1],get_pos[2],get_org[3],get_org[4],get_org[5]]
                        $ 477 "pre_tp≔tilt_2f_fun(get_pos,[0,0], False , True )"
                        global pre_tp=tilt_2f_fun(get_pos,[0,0],  False  ,  True  )
                      end
                    end
                  end
                end
                $ 478 "A_Prepos_l[move_i]=pre_tp"
                A_Prepos_l[move_i]=pre_tp
              end
              $ 479 "move_i≔move_i+1"
              global move_i=move_i+1
            end
            $ 480 "homeing()"
            homeing()
            $ 481 "Wait read_port_register(170)≟1"
            while (not( read_port_register (170) == 1)):
              sync()
            end
            $ 482 "write_port_register(170,0)"
            write_port_register(170,0)
          else:
            $ 483 "Else" "noBreak"
            $ 484 "value from pendant"
            $ 485 "move_i≔1"
            global move_i=1
            $ 487 "Touch_FrontandSide"
            $ 488 "If EXT_flag1[11]≟ True "
            if (EXT_flag1[11] ==   True  ):
              $ 489 "Touch front and side_Right"
              $ 490 "move_center≔pose_add(first_p_wp, p[-first_p_wp[0]+(get_center-work_touch_dis)/1000,0,0,0,0,0])"
              global move_center= pose_add (first_p_wp, p[-first_p_wp[0]+(get_center-work_touch_dis)/1000,0,0,0,0,0])
              $ 491 "get_pose_side_t≔0"
              global get_pose_side_t=0
              $ 493 "move_center[2]=(center_height+a7_cell_bottom)/1000"
              move_center[2]=(center_height+a7_cell_bottom)/1000
              $ 495 "MoveL"
              $ 496 "move_center" "breakAfter"
              movel(pose_trans(Base, move_center), a=0.5, v=0.15)
              $ 497 "touch_center≔contact_fun(p[0,0,0,0,0,0],[1,0,0],20000,20,20)"
              global touch_center=contact_fun(p[0,0,0,0,0,0],[1,0,0],20000,20,20)
              $ 498 "direction(p[0,0,0,0,0,0],[-1,0,0],10,180,200)"
              direction(p[0,0,0,0,0,0],[-1,0,0],10,180,200)
              $ 499 "get_center≔touch_center[0]*1000"
              global get_center=touch_center[0]*1000
              $ 500 "a7_f_distance≔get_center"
              global a7_f_distance=get_center
              $ 501 "move_center≔pose_add(move_center,p[0,sec_touch_dis/1000,0,0,0,0])"
              global move_center= pose_add (move_center,p[0,sec_touch_dis/1000,0,0,0,0])
              $ 502 "move_center[0]=touch_center[0]-20/1000"
              move_center[0]=touch_center[0]-20/1000
              $ 503 "MoveL"
              $ 504 "move_center" "breakAfter"
              movel(pose_trans(Base, move_center), a=0.5, v=0.15)
              $ 505 "touch_center2≔contact_fun(p[0,0,0,0,0,0],[1,0,0],20000,20,20)"
              global touch_center2=contact_fun(p[0,0,0,0,0,0],[1,0,0],20000,20,20)
              $ 506 "center_line≔get_feature_Line(touch_center,touch_center2)"
              global center_line=get_feature_Line(touch_center,touch_center2)
              $ 507 "event_cal_on≔ True "
              global event_cal_on=  True
              $ 508 "direction(p[0,0,0,0,0,0],[-1,0,0],10,180,200)"
              direction(p[0,0,0,0,0,0],[-1,0,0],10,180,200)
              $ 510 "homeing()"
              homeing()
              $ 511 "b2_left_par≔ False "
              global b2_left_par=  False
              $ 512 "b8_wv_2f≔ False "
              global b8_wv_2f=  False
              $ 513 "b2_cell≔b1_cell_info_R"
              global b2_cell=b1_cell_info_R
              $ 514 "get_pos≔get_lr(side_p_R,a6_f_width,[35,0,0,0,0],a7_f_distance,b2_left_par,b8_wv_2f,Touch_dis,get_margin_z,get_pose_side_t,30,0,center_line, True )"
              global get_pos=get_lr(p[.471584857321, -.427242166643, .026448165242, 1.806736638758, -1.227818761912, 1.383474453522],a6_f_width,[35,0,0,0,0],a7_f_distance,b2_left_par,b8_wv_2f,Touch_dis,get_margin_z,get_pose_side_t,30,0,center_line,  True  )
              $ 516 "pre_tp≔get_pos"
              global pre_tp=get_pos
              $ 517 "pre_tp≔pose_add(pre_tp, p[side_pos_x/1000,0,0,0,0,0])"
              global pre_tp= pose_add (pre_tp, p[side_pos_x/1000,0,0,0,0,0])
              $ 518 "pre_tp[2]=(center_height+a7_cell_bottom)/1000"
              pre_tp[2]=(center_height+a7_cell_bottom)/1000
              $ 519 "MoveL"
              $ 520 "pre_tp" "breakAfter"
              movel(pose_trans(Base, pre_tp), a=0.8, v=0.4)
              $ 521 "touch_side≔contact_fun(p[0,0,0,0,0,0],[0,-1,0],20000,13,13)"
              global touch_side=contact_fun(p[0,0,0,0,0,0],[0,-1,0],20000,13,13)
              $ 522 "touch_side≔get_feature_pose(touch_side,center_line)"
              global touch_side=get_feature_pose(touch_side,center_line)
              $ 523 "direction(p[0,0,0,0,0,0],[0,1,0],10,180,200)"
              direction(p[0,0,0,0,0,0],[0,1,0],10,180,200)
              $ 524 "write_welder(4, False )"
              write_welder(4,  False  )
              $ 525 "get_pose_side_t≔touch_side[1]*1000"
              global get_pose_side_t=touch_side[1]*1000
              $ 526 "get_pose_side_t≔get_pose_side_t+(a6_f_width/2)"
              global get_pose_side_t=get_pose_side_t+(a6_f_width/2)
              $ 527 "event_side_on≔ True "
              global event_side_on=  True
              $ 528 "MoveL"
              $ 529 "Direction: Base"
              global move_thread_flag_529=0
              thread move_thread_529():
                enter_critical
                move_thread_flag_529 = 1
                local towardsPos=calculate_point_to_move_towards(p[0.0,0.0,0.0,0.0,0.0,0.0], [-1,1,0], 0.03)
                movel(towardsPos, a=0.3, v=0.15)
                move_thread_flag_529 = 2
                exit_critical
              end
              move_thread_flag_529 = 0
              move_thread_han_529 = run move_thread_529()
              while (True):
                sleep(1.0E-10)
                if (move_thread_flag_529 > 1):
                  join move_thread_han_529
                  $ 530 "Until (distance)"
                  break
                end
                sync()
              end
              $ 531 "homeing()"
              homeing()
            else:
              $ 532 "Else" "noBreak"
              $ 533 "Touch front and side_Left"
              $ 534 "move_center≔pose_add(first_p_wp, p[-first_p_wp[0]+(get_center-work_touch_dis)/1000,0,0,0,0,0])"
              global move_center= pose_add (first_p_wp, p[-first_p_wp[0]+(get_center-work_touch_dis)/1000,0,0,0,0,0])
              $ 535 "get_pose_side_t≔0"
              global get_pose_side_t=0
              $ 537 "move_center[2]=(center_height+a7_cell_bottom)/1000"
              move_center[2]=(center_height+a7_cell_bottom)/1000
              $ 539 "MoveL"
              $ 540 "move_center" "breakAfter"
              movel(pose_trans(Base, move_center), a=0.5, v=0.15)
              $ 541 "touch_center≔contact_fun(p[0,0,0,0,0,0],[1,0,0],20000,20,20)"
              global touch_center=contact_fun(p[0,0,0,0,0,0],[1,0,0],20000,20,20)
              $ 542 "direction(p[0,0,0,0,0,0],[-1,0,0],10,180,200)"
              direction(p[0,0,0,0,0,0],[-1,0,0],10,180,200)
              $ 543 "get_center≔touch_center[0]*1000"
              global get_center=touch_center[0]*1000
              $ 544 "a7_f_distance≔get_center"
              global a7_f_distance=get_center
              $ 545 "move_center≔pose_add(move_center,p[0,sec_touch_dis/1000,0,0,0,0])"
              global move_center= pose_add (move_center,p[0,sec_touch_dis/1000,0,0,0,0])
              $ 546 "move_center[0]=touch_center[0]-20/1000"
              move_center[0]=touch_center[0]-20/1000
              $ 547 "MoveL"
              $ 548 "move_center" "breakAfter"
              movel(pose_trans(Base, move_center), a=0.5, v=0.15)
              $ 549 "touch_center2≔contact_fun(p[0,0,0,0,0,0],[1,0,0],20000,20,20)"
              global touch_center2=contact_fun(p[0,0,0,0,0,0],[1,0,0],20000,20,20)
              $ 550 "center_line≔get_feature_Line(touch_center,touch_center2)"
              global center_line=get_feature_Line(touch_center,touch_center2)
              $ 551 "event_cal_on≔ True "
              global event_cal_on=  True
              $ 552 "direction(p[0,0,0,0,0,0],[-1,0,0],10,180,200)"
              direction(p[0,0,0,0,0,0],[-1,0,0],10,180,200)
              $ 554 "homeing()"
              homeing()
              $ 555 "b2_left_par≔ True "
              global b2_left_par=  True
              $ 556 "b8_wv_2f≔ False "
              global b8_wv_2f=  False
              $ 557 "b2_cell≔b1_cell_info_L"
              global b2_cell=b1_cell_info_L
              $ 558 "get_pos≔get_lr(side_p_L,a6_f_width,[35,0,0,0,0],a7_f_distance,b2_left_par,b8_wv_2f,Touch_dis,get_margin_z,get_pose_side_t,30,0,center_line, True )"
              global get_pos=get_lr(p[.411215372122, .375785944375, -.010176539343, -1.953488355698, -1.125710367676, -1.228829273458],a6_f_width,[35,0,0,0,0],a7_f_distance,b2_left_par,b8_wv_2f,Touch_dis,get_margin_z,get_pose_side_t,30,0,center_line,  True  )
              $ 560 "pre_tp≔get_pos"
              global pre_tp=get_pos
              $ 561 "pre_tp≔pose_add(pre_tp, p[side_pos_x/1000,0,0,0,0,0])"
              global pre_tp= pose_add (pre_tp, p[side_pos_x/1000,0,0,0,0,0])
              $ 562 "pre_tp[2]=(center_height+a7_cell_bottom)/1000"
              pre_tp[2]=(center_height+a7_cell_bottom)/1000
              $ 563 "MoveL"
              $ 564 "pre_tp" "breakAfter"
              movel(pose_trans(Base, pre_tp), a=0.8, v=0.4)
              $ 565 "touch_side≔contact_fun(p[0,0,0,0,0,0],[0,1,0],20000,13,13)"
              global touch_side=contact_fun(p[0,0,0,0,0,0],[0,1,0],20000,13,13)
              $ 566 "touch_side≔get_feature_pose(touch_side,center_line)"
              global touch_side=get_feature_pose(touch_side,center_line)
              $ 567 "direction(p[0,0,0,0,0,0],[0,-1,0],10,180,200)"
              direction(p[0,0,0,0,0,0],[0,-1,0],10,180,200)
              $ 568 "write_welder(4, False )"
              write_welder(4,  False  )
              $ 569 "get_pose_side_t≔touch_side[1]*1000"
              global get_pose_side_t=touch_side[1]*1000
              $ 570 "get_pose_side_t≔get_pose_side_t-(a6_f_width/2)"
              global get_pose_side_t=get_pose_side_t-(a6_f_width/2)
              $ 571 "event_side_on≔ True "
              global event_side_on=  True
              $ 572 "MoveL"
              $ 573 "Direction: Base"
              global move_thread_flag_573=0
              thread move_thread_573():
                enter_critical
                move_thread_flag_573 = 1
                local towardsPos=calculate_point_to_move_towards(p[0.0,0.0,0.0,0.0,0.0,0.0], [-1,-1,0], 0.03)
                movel(towardsPos, a=0.3, v=0.15)
                move_thread_flag_573 = 2
                exit_critical
              end
              move_thread_flag_573 = 0
              move_thread_han_573 = run move_thread_573()
              while (True):
                sleep(1.0E-10)
                if (move_thread_flag_573 > 1):
                  join move_thread_han_573
                  $ 574 "Until (distance)"
                  break
                end
                sync()
              end
              $ 575 "homeing()"
              homeing()
            end
            $ 577 "Wait event_side_on≟ False "
            while (not(event_side_on ==   False  )):
              sync()
            end
          end
          $ 578 "move and touch"
          $ 579 "Touch Move"
          $ 580 "HOR_L"
          $ 581 "If A_Prepos_l[A_HOR]≠p[0,0,0,0,0,0]"
          if (A_Prepos_l[A_HOR] != p[0,0,0,0,0,0]):
            $ 582 "b2_left_par≔ True "
            global b2_left_par=  True
            $ 583 "b8_wv_2f≔ True "
            global b8_wv_2f=  True
            $ 584 "b7_tilt_degree≔[0,0,0]"
            global b7_tilt_degree=[0,0,0]
            $ 585 "A_sel_v≔A_HOR"
            global A_sel_v=A_HOR
            $ 586 "wv_direction≔1"
            global wv_direction=1
            $ 587 "Call MoveandTouchFun_2f"
            MoveandTouchFun_2f()
            $ 588 "If b1_cell_info_L≟A or b1_cell_info_L≟C or b1_cell_info_L≟c"
            if (b1_cell_info_L == A  or  b1_cell_info_L == C  or  b1_cell_info_L == c):
              $ 589 "If A_Prepos_l[A_VL1]≟p[0,0,0,0,0,0]"
              if (A_Prepos_l[A_VL1] == p[0,0,0,0,0,0]):
                $ 591 "g_tp≔A_Prepos_l[A_HOR]"
                global g_tp=A_Prepos_l[A_HOR]
                $ 594 "Folder"
                $ 595 "g_cp≔get_actual_tcp_pose()"
                global g_cp= get_actual_tcp_pose ()
                $ 596 "g_cp≔pose_trans(g_cp, p[0,0,0,d2r(12),d2r(5),0])"
                global g_cp= pose_trans (g_cp, p[0,0,0,d2r(12),d2r(5),0])
                $ 597 "MoveL"
                $ 598 "g_cp" "breakAfter"
                movel(pose_trans(Base, g_cp), a=0.08, v=0.08)
                $ 599 "for_x_HOR≔contact_fun(A_Touch_p[A_sel_v],[-1*wv_direction,0,0],10000,15,15,  False)"
                global for_x_HOR=contact_fun(A_Touch_p[A_sel_v],[-1*wv_direction,0,0],10000,15,15,  False)
                $ 600 "direction(p[0,0,0,0,0,0],[0,-1,0],20,120,160)"
                direction(p[0,0,0,0,0,0],[0,-1,0],20,120,160)
                $ 601 "write_welder(4, False )"
                write_welder(4,  False  )
              else:
                $ 602 "Else" "noBreak"
                $ 603 "for_x_HOR≔p[0,0,0,0,0,0]"
                global for_x_HOR=p[0,0,0,0,0,0]
              end
            end
            $ 611 "If point_dist(A_Prepos_l[A_HOR], A_Prepos_l[A_VL1])>0.032"
            if (point_dist(A_Prepos_l[A_HOR], A_Prepos_l[A_VL1])>0.032):
              $ 612 "homeing()"
              homeing()
            end
          end
          $ 613 "VL1"
          $ 614 "If A_Prepos_l[A_VL1]≠p[0,0,0,0,0,0]"
          if (A_Prepos_l[A_VL1] != p[0,0,0,0,0,0]):
            $ 615 "b2_left_par≔ True "
            global b2_left_par=  True
            $ 616 "b8_wv_2f≔ False "
            global b8_wv_2f=  False
            $ 617 "b7_tilt_degree≔[0,0,0]"
            global b7_tilt_degree=[0,0,0]
            $ 618 "A_sel_v≔A_VL1"
            global A_sel_v=A_VL1
            $ 619 "A_sel_v_end≔A_VL1_END"
            global A_sel_v_end=A_VL1_END
            $ 620 "b2_par_cd≔0"
            global b2_par_cd=0
            $ 621 "If b1_cell_info_L≟A or b1_cell_info_L≟C or b1_cell_info_L≟c"
            if (b1_cell_info_L == A  or  b1_cell_info_L == C  or  b1_cell_info_L == c):
              $ 622 "Scallup_check≔ True "
              global Scallup_check=  True
            else:
              $ 623 "Else" "noBreak"
              $ 624 "Scallup_check≔ False "
              global Scallup_check=  False
            end
            $ 625 "Call MoveandTouchFun_3f"
            MoveandTouchFun_3f()
            $ 626 "If b1_cell_info_L≟A or b1_cell_info_L≟C or b1_cell_info_L≟c"
            if (b1_cell_info_L == A  or  b1_cell_info_L == C  or  b1_cell_info_L == c):
              $ 627 "If A_Prepos_l[A_HOR]≟p[0,0,0,0,0,0]"
              if (A_Prepos_l[A_HOR] == p[0,0,0,0,0,0]):
                $ 628 "direction(p[0,0,0,0,0,0],[0,-1,0],8,120,160)"
                direction(p[0,0,0,0,0,0],[0,-1,0],8,120,160)
                $ 630 "AAgcp≔get_actual_tcp_pose()"
                global AAgcp= get_actual_tcp_pose ()
                $ 631 "AAgangle≔up_left"
                global AAgangle=p[.492775857339, .409517380626, -.029063830209, -2.419264859926, -.998084331190, -1.368689080860]
                $ 632 "AAgtp≔p[AAgcp[0],AAgcp[1],AAgcp[2],AAgangle[3],AAgangle[4],AAgangle[5]]"
                global AAgtp=p[AAgcp[0],AAgcp[1],AAgcp[2],AAgangle[3],AAgangle[4],AAgangle[5]]
                $ 633 "MoveL"
                $ 634 "AAgtp" "breakAfter"
                movel(pose_trans(Base, AAgtp), a=0.08, v=0.08)
                $ 636 "for_z_VL1≔contact_fun(p[0,0,0,0,0,0],[0,0,-1],10000,15,15,  False)"
                global for_z_VL1=contact_fun(p[0,0,0,0,0,0],[0,0,-1],10000,15,15,  False)
                $ 637 "direction(p[0,0,0,0,0,0],[0,0,1],20,120,160)"
                direction(p[0,0,0,0,0,0],[0,0,1],20,120,160)
                $ 638 "write_welder(4, False )"
                write_welder(4,  False  )
              else:
                $ 639 "Else" "noBreak"
                $ 640 "for_z_VL1≔p[0,0,0,0,0,0]"
                global for_z_VL1=p[0,0,0,0,0,0]
              end
            end
          end
          $ 641 "HOR_ML"
          $ 642 "If A_Prepos_l[A_HOR_ML]≠p[0,0,0,0,0,0]"
          if (A_Prepos_l[A_HOR_ML] != p[0,0,0,0,0,0]):
            $ 643 "b2_left_par≔ True "
            global b2_left_par=  True
            $ 644 "b8_wv_2f≔ True "
            global b8_wv_2f=  True
            $ 645 "b7_tilt_degree≔[0,0,0]"
            global b7_tilt_degree=[0,0,0]
            $ 646 "A_sel_v≔A_HOR_ML"
            global A_sel_v=A_HOR_ML
            $ 647 "If b1_cell_info_L≟C or b1_cell_info_L≟D"
            if (b1_cell_info_L == C  or  b1_cell_info_L == D):
              $ 648 "wv_direction≔1"
              global wv_direction=1
              $ 649 "Call MoveFun"
              MoveFun()
              $ 650 "for_cal_xy≔contact_fun(p[0,0,0,0,0,0],[1,0,0],20000,20,20)"
              global for_cal_xy=contact_fun(p[0,0,0,0,0,0],[1,0,0],20000,20,20)
              $ 651 "direction(p[0,0,0,0,0,0],[-1,0,0],15,120,160)"
              direction(p[0,0,0,0,0,0],[-1,0,0],15,120,160)
              $ 652 "direction(p[0,0,0,0,0,0],[0,-1,0],60,120,160)"
              direction(p[0,0,0,0,0,0],[0,-1,0],60,120,160)
              $ 653 "direction(p[0,0,0,0,0,0],[1,0,0],20,120,160)"
              direction(p[0,0,0,0,0,0],[1,0,0],20,120,160)
              $ 654 "for_cal_x_wel≔contact_fun(p[0,0,0,0,0,0],[0,1,0],20000,20,20)"
              global for_cal_x_wel=contact_fun(p[0,0,0,0,0,0],[0,1,0],20000,20,20)
              $ 655 "direction(p[0,0,0,0,0,0],[0,-1,0],20,120,160)"
              direction(p[0,0,0,0,0,0],[0,-1,0],20,120,160)
              $ 656 "for_cal_y_wel≔contact_fun(p[0,0,0,0,0,0],[1,0,0],20000,20,20)"
              global for_cal_y_wel=contact_fun(p[0,0,0,0,0,0],[1,0,0],20000,20,20)
              $ 657 "direction(p[0,0,0,0,0,0],[-1,0,0],20,120,160)"
              direction(p[0,0,0,0,0,0],[-1,0,0],20,120,160)
              $ 658 "for_z_VLR2≔contact_fun(p[0,0,0,0,0,0],[0,0,-1],20000,20,20)"
              global for_z_VLR2=contact_fun(p[0,0,0,0,0,0],[0,0,-1],20000,20,20)
              $ 659 "direction(p[0,0,0,0,0,0],[0,0,1],20,120,160)"
              direction(p[0,0,0,0,0,0],[0,0,1],20,120,160)
              $ 660 "for_cal_rot≔A_Touch_p[A_HOR]"
              global for_cal_rot=A_Touch_p[A_HOR]
              $ 661 "A_Touch_p[A_sel_v]=p[for_cal_xy[0],for_cal_xy[1],for_z_VLR2[2],for_cal_rot[3],for_cal_rot[4],for_cal_rot[5]]"
              A_Touch_p[A_sel_v]=p[for_cal_xy[0],for_cal_xy[1],for_z_VLR2[2],for_cal_rot[3],for_cal_rot[4],for_cal_rot[5]]
              $ 662 "A_Touch_p[A_sel_v]=pose_trans(A_Touch_p[A_sel_v], p[Touch_dis/1000,0,0,0,0,0])"
              A_Touch_p[A_sel_v]= pose_trans (A_Touch_p[A_sel_v], p[Touch_dis/1000,0,0,0,0,0])
              $ 663 "write_welder(4, False )"
              write_welder(4,  False  )
            else:
              $ 664 "Else" "noBreak"
              $ 665 "wv_direction≔1"
              global wv_direction=1
              $ 666 "for_cal_rot≔A_Touch_p[A_HOR]"
              global for_cal_rot=A_Touch_p[A_HOR]
              $ 667 "Call MoveFun_cd"
              MoveFun_cd()
              $ 668 "for_cal_y_wel≔contact_fun(p[0,0,0,0,0,0],[1,0,0],20000,20,20)"
              global for_cal_y_wel=contact_fun(p[0,0,0,0,0,0],[1,0,0],20000,20,20)
              $ 669 "for_cal_y_wel[2]=for_cal_rot[2]"
              for_cal_y_wel[2]=for_cal_rot[2]
              $ 670 "dir_x_cal≔get_feature_Line(for_cal_rot,for_cal_y_wel)"
              global dir_x_cal=get_feature_Line(for_cal_rot,for_cal_y_wel)
              $ 671 "direction(p[0,0,0,0,0,0],[-1,0,0],40,120,160)"
              direction(p[0,0,0,0,0,0],[-1,0,0],40,120,160)
              $ 672 "direction(p[0,0,0,0,0,0],[0,-1,0],80,120,160)"
              direction(p[0,0,0,0,0,0],[0,-1,0],80,120,160)
              $ 673 "for_cal_y_wel≔contact_fun(p[0,0,0,0,0,0],[1,0,0],20000,20,20)"
              global for_cal_y_wel=contact_fun(p[0,0,0,0,0,0],[1,0,0],20000,20,20)
              $ 674 "direction(p[0,0,0,0,0,0],[-1,0,0],5,120,160)"
              direction(p[0,0,0,0,0,0],[-1,0,0],5,120,160)
              $ 675 "direction(p[0,0,0,0,0,0],[0,1,0],60,120,160)"
              direction(p[0,0,0,0,0,0],[0,1,0],60,120,160)
              $ 676 "direction(p[0,0,0,0,0,0],[1,0,0],7,120,160)"
              direction(p[0,0,0,0,0,0],[1,0,0],7,120,160)
              $ 677 "for_cal_x_wel≔contact_fun(p[0,0,0,0,0,0],[0,-1,0],20000,20,20)"
              global for_cal_x_wel=contact_fun(p[0,0,0,0,0,0],[0,-1,0],20000,20,20)
              $ 678 "get_ml≔get_feature_pose(for_cal_x_wel,for_cal_rot)"
              global get_ml=get_feature_pose(for_cal_x_wel,for_cal_rot)
              $ 680 "A_Touch_p[A_sel_v]=feature_offset(for_cal_rot,p[0,get_ml[0]+(-cd_offset+cd_extra_dis)/1000,0,0,0,0],dir_x_cal)"
              A_Touch_p[A_sel_v]=feature_offset(for_cal_rot,p[0,get_ml[0]+(-cd_offset+cd_extra_dis)/1000,0,0,0,0],dir_x_cal)
              $ 681 "direction(p[0,0,0,0,0,0],[0,1,0],5,120,160)"
              direction(p[0,0,0,0,0,0],[0,1,0],5,120,160)
              $ 682 "direction(p[0,0,0,0,0,0],[-1,0,0],20,120,160)"
              direction(p[0,0,0,0,0,0],[-1,0,0],20,120,160)
              $ 683 "write_welder(4, False )"
              write_welder(4,  False  )
            end
            $ 684 "homeing()"
            homeing()
          else:
            $ 685 "Else" "noBreak"
            $ 686 "homeing()"
            homeing()
          end
          $ 687 "VL2"
          $ 688 "If A_Prepos_l[A_VL2]≠p[0,0,0,0,0,0]"
          if (A_Prepos_l[A_VL2] != p[0,0,0,0,0,0]):
            $ 689 "b2_left_par≔ True "
            global b2_left_par=  True
            $ 690 "b8_wv_2f≔ False "
            global b8_wv_2f=  False
            $ 691 "b7_tilt_degree≔basic_tilt_3f"
            global b7_tilt_degree=basic_tilt_3f
            $ 692 "A_sel_v≔A_VL2"
            global A_sel_v=A_VL2
            $ 693 "A_sel_v_end≔A_VL2_END"
            global A_sel_v_end=A_VL2_END
            $ 694 "b2_par_cd≔1"
            global b2_par_cd=1
            $ 695 "If b1_cell_info_L≟A or b1_cell_info_L≟C or b1_cell_info_L≟c"
            if (b1_cell_info_L == A  or  b1_cell_info_L == C  or  b1_cell_info_L == c):
              $ 696 "Scallup_check≔ True "
              global Scallup_check=  True
            else:
              $ 697 "Else" "noBreak"
              $ 698 "Scallup_check≔ False "
              global Scallup_check=  False
            end
            $ 699 "If b1_cell_info_L≟d or b1_cell_info_L≟c"
            if (b1_cell_info_L == d  or  b1_cell_info_L == c):
              $ 700 "Halt"
              halt
            else:
              $ 701 "Else" "noBreak"
              $ 702 "If A_Touch_p[A_VL1]≟p[0,0,0,0,0,0]"
              if (A_Touch_p[A_VL1] == p[0,0,0,0,0,0]):
                $ 703 "Call MoveandTouchFun_3f"
                MoveandTouchFun_3f()
                $ 704 "If A_Prepos_l[A_HOR_ML]≟p[0,0,0,0,0,0]"
                if (A_Prepos_l[A_HOR_ML] == p[0,0,0,0,0,0]):
                  $ 705 "direction(p[0,0,0,0,0,0],[-1,-1,0],8,120,160)"
                  direction(p[0,0,0,0,0,0],[-1,-1,0],8,120,160)
                  $ 706 "AAgcp≔get_actual_tcp_pose()"
                  global AAgcp= get_actual_tcp_pose ()
                  $ 707 "AAgangle≔up_left"
                  global AAgangle=p[.492775857339, .409517380626, -.029063830209, -2.419264859926, -.998084331190, -1.368689080860]
                  $ 708 "AAgtp≔p[AAgcp[0],AAgcp[1],AAgcp[2],AAgangle[3],AAgangle[4],AAgangle[5]]"
                  global AAgtp=p[AAgcp[0],AAgcp[1],AAgcp[2],AAgangle[3],AAgangle[4],AAgangle[5]]
                  $ 709 "MoveL"
                  $ 710 "AAgtp" "breakAfter"
                  movel(pose_trans(Base, AAgtp), a=0.08, v=0.08)
                  $ 712 "for_z_VLR2≔contact_fun(p[0,0,0,0,0,0],[0,0,-1],20000,20,20)"
                  global for_z_VLR2=contact_fun(p[0,0,0,0,0,0],[0,0,-1],20000,20,20)
                  $ 713 "direction(p[0,0,0,0,0,0],[0,0,1],10,120,160)"
                  direction(p[0,0,0,0,0,0],[0,0,1],10,120,160)
                end
                $ 714 "touch_tmp≔A_Touch_p[A_sel_v]"
                global touch_tmp=A_Touch_p[A_sel_v]
                $ 715 "touch_tmp[2]=for_z_VLR2[2]"
                touch_tmp[2]=for_z_VLR2[2]
                $ 716 "A_Touch_p[A_sel_v]=touch_tmp"
                A_Touch_p[A_sel_v]=touch_tmp
                $ 717 "for_cal_y_wel≔A_Touch_p[A_sel_v]"
                global for_cal_y_wel=A_Touch_p[A_sel_v]
                $ 718 "for_cal_x_wel≔A_Touch_p[A_sel_v]"
                global for_cal_x_wel=A_Touch_p[A_sel_v]
              else:
                $ 719 "Else" "noBreak"
                $ 720 "If A_Prepos_l[A_HOR_ML]≟p[0,0,0,0,0,0]"
                if (A_Prepos_l[A_HOR_ML] == p[0,0,0,0,0,0]):
                  $ 721 "Call MoveFun"
                  MoveFun()
                  $ 722 "for_cal_y_wel≔contact_fun(p[0,0,0,0,0,0],[1,0,0],20000,20,20)"
                  global for_cal_y_wel=contact_fun(p[0,0,0,0,0,0],[1,0,0],20000,20,20)
                  $ 723 "direction(p[0,0,0,0,0,0],[-1,0,0],40,120,160)"
                  direction(p[0,0,0,0,0,0],[-1,0,0],40,120,160)
                  $ 724 "direction(p[0,0,0,0,0,0],[0,1,0],60,120,160)"
                  direction(p[0,0,0,0,0,0],[0,1,0],60,120,160)
                  $ 725 "var_2≔contact_fun(p[0,0,0,0,0,0],[1,0,0],20000,20,20)"
                  global var_2=contact_fun(p[0,0,0,0,0,0],[1,0,0],20000,20,20)
                  $ 726 "direction(p[0,0,0,0,0,0],[-1,0,0],5,120,160)"
                  direction(p[0,0,0,0,0,0],[-1,0,0],5,120,160)
                  $ 727 "direction(p[0,0,0,0,0,0],[0,-1,0],60,120,160)"
                  direction(p[0,0,0,0,0,0],[0,-1,0],60,120,160)
                  $ 728 "direction(p[0,0,0,0,0,0],[1,0,0],10,120,160)"
                  direction(p[0,0,0,0,0,0],[1,0,0],10,120,160)
                  $ 729 "for_cal_x_wel≔contact_fun(p[0,0,0,0,0,0],[0,1,0],20000,20,20)"
                  global for_cal_x_wel=contact_fun(p[0,0,0,0,0,0],[0,1,0],20000,20,20)
                  $ 730 "direction(p[0,0,0,0,0,0],[0,-1,0],20,120,160)"
                  direction(p[0,0,0,0,0,0],[0,-1,0],20,120,160)
                  $ 731 "AAgcp≔get_actual_tcp_pose()"
                  global AAgcp= get_actual_tcp_pose ()
                  $ 732 "AAgangle≔up_left"
                  global AAgangle=p[.492775857339, .409517380626, -.029063830209, -2.419264859926, -.998084331190, -1.368689080860]
                  $ 733 "AAgtp≔p[AAgcp[0],AAgcp[1],AAgcp[2],AAgangle[3],AAgangle[4],AAgangle[5]]"
                  global AAgtp=p[AAgcp[0],AAgcp[1],AAgcp[2],AAgangle[3],AAgangle[4],AAgangle[5]]
                  $ 734 "MoveL"
                  $ 735 "AAgtp" "breakAfter"
                  movel(pose_trans(Base, AAgtp), a=0.08, v=0.08)
                  $ 737 "for_z_VLR2≔contact_fun(p[0,0,0,0,0,0],[0,0,-1],20000,20,20)"
                  global for_z_VLR2=contact_fun(p[0,0,0,0,0,0],[0,0,-1],20000,20,20)
                  $ 738 "direction(p[0,0,0,0,0,0],[0,0,1],10,120,160)"
                  direction(p[0,0,0,0,0,0],[0,0,1],10,120,160)
                  $ 739 "direction(p[0,0,0,0,0,0],[-1,0,0],20,120,160)"
                  direction(p[0,0,0,0,0,0],[-1,0,0],20,120,160)
                end
                $ 740 "for_cal_rot≔A_Touch_p[A_VL1]"
                global for_cal_rot=A_Touch_p[A_VL1]
                $ 741 "touch_tmp=p[for_cal_y_wel[0],for_cal_x_wel[1],for_cal_x_wel[2],for_cal_rot[3],for_cal_rot[4],for_cal_rot[5]]"
                touch_tmp=p[for_cal_y_wel[0],for_cal_x_wel[1],for_cal_x_wel[2],for_cal_rot[3],for_cal_rot[4],for_cal_rot[5]]
                $ 742 "If Scallup_check≟ False "
                if (Scallup_check ==   False  ):
                  $ 743 "touch_tmp≔pose_trans(touch_tmp,p[-(Touch_dis)/1000,0,0,0,0,0])"
                  global touch_tmp= pose_trans (touch_tmp,p[-(Touch_dis)/1000,0,0,0,0,0])
                else:
                  $ 744 "Else" "noBreak"
                  $ 745 "Scallup_check≔ False "
                  global Scallup_check=  False
                end
                $ 746 "A_Touch_p[A_sel_v]=touch_tmp"
                A_Touch_p[A_sel_v]=touch_tmp
                $ 747 "write_welder(4, False )"
                write_welder(4,  False  )
              end
            end
            $ 748 "b2_par_cd≔0"
            global b2_par_cd=0
            $ 749 "homeing()"
            homeing()
          else:
            $ 750 "Else" "noBreak"
            $ 751 "homeing()"
            homeing()
          end
          $ 752 "HOR_R"
          $ 753 "If A_Prepos_l[A_HOR_R]≠p[0,0,0,0,0,0]"
          if (A_Prepos_l[A_HOR_R] != p[0,0,0,0,0,0]):
            $ 754 "b2_left_par≔ False "
            global b2_left_par=  False
            $ 755 "b8_wv_2f≔ True "
            global b8_wv_2f=  True
            $ 756 "b7_tilt_degree≔[0,0,0]"
            global b7_tilt_degree=[0,0,0]
            $ 757 "A_sel_v≔A_HOR_R"
            global A_sel_v=A_HOR_R
            $ 758 "wv_direction≔-1"
            global wv_direction=-1
            $ 759 "Call MoveandTouchFun_2f"
            MoveandTouchFun_2f()
            $ 761 "If b1_cell_info_R≟A or b1_cell_info_R≟C or b1_cell_info_R≟c"
            if (b1_cell_info_R == A  or  b1_cell_info_R == C  or  b1_cell_info_R == c):
              $ 762 "If A_Prepos_l[A_VR1]≟p[0,0,0,0,0,0]"
              if (A_Prepos_l[A_VR1] == p[0,0,0,0,0,0]):
                $ 764 "g_tp≔A_Prepos_l[A_HOR_R]"
                global g_tp=A_Prepos_l[A_HOR_R]
                $ 765 "Folder"
                $ 766 "g_cp≔get_actual_tcp_pose()"
                global g_cp= get_actual_tcp_pose ()
                $ 767 "g_cp≔pose_trans(g_cp, p[0,0,0,d2r(-12),d2r(5),0])"
                global g_cp= pose_trans (g_cp, p[0,0,0,d2r(-12),d2r(5),0])
                $ 768 "MoveL"
                $ 769 "g_cp" "breakAfter"
                movel(pose_trans(Base, g_cp), a=0.08, v=0.08)
                $ 772 "for_x_HOR_R≔contact_fun(A_Touch_p[A_HOR_R],[-1*wv_direction,0,0],10000,15,15,  False)"
                global for_x_HOR_R=contact_fun(A_Touch_p[A_HOR_R],[-1*wv_direction,0,0],10000,15,15,  False)
                $ 773 "direction(p[0,0,0,0,0,0],[0,1,0],20,120,160)"
                direction(p[0,0,0,0,0,0],[0,1,0],20,120,160)
                $ 774 "write_welder(4, False )"
                write_welder(4,  False  )
              else:
                $ 775 "Else" "noBreak"
                $ 776 "for_x_HOR_R≔p[0,0,0,0,0,0]"
                global for_x_HOR_R=p[0,0,0,0,0,0]
              end
            end
            $ 777 "wv_direction≔1"
            global wv_direction=1
            $ 778 "If point_dist(A_Prepos_l[A_HOR_R], A_Prepos_l[A_VR1])>0.0327"
            if (point_dist(A_Prepos_l[A_HOR_R], A_Prepos_l[A_VR1])>0.0327):
              $ 779 "homeing()"
              homeing()
            end
          end
          $ 780 "VR1"
          $ 781 "If A_Prepos_l[A_VR1]≠p[0,0,0,0,0,0]"
          if (A_Prepos_l[A_VR1] != p[0,0,0,0,0,0]):
            $ 782 "b2_left_par≔ False "
            global b2_left_par=  False
            $ 783 "b8_wv_2f≔ False "
            global b8_wv_2f=  False
            $ 784 "b7_tilt_degree≔basic_tilt_3f"
            global b7_tilt_degree=basic_tilt_3f
            $ 785 "A_sel_v≔A_VR1"
            global A_sel_v=A_VR1
            $ 786 "A_sel_v_end≔A_VR1_END"
            global A_sel_v_end=A_VR1_END
            $ 787 "b2_par_cd≔0"
            global b2_par_cd=0
            $ 788 "If b1_cell_info_R≟A or b1_cell_info_R≟C or b1_cell_info_R≟c"
            if (b1_cell_info_R == A  or  b1_cell_info_R == C  or  b1_cell_info_R == c):
              $ 789 "Scallup_check≔ True "
              global Scallup_check=  True
            else:
              $ 790 "Else" "noBreak"
              $ 791 "Scallup_check≔ False "
              global Scallup_check=  False
            end
            $ 792 "Call MoveandTouchFun_3f"
            MoveandTouchFun_3f()
            $ 793 "If b1_cell_info_R≟A or b1_cell_info_R≟C or b1_cell_info_R≟c"
            if (b1_cell_info_R == A  or  b1_cell_info_R == C  or  b1_cell_info_R == c):
              $ 794 "If A_Prepos_l[A_HOR_R]≟p[0,0,0,0,0,0]"
              if (A_Prepos_l[A_HOR_R] == p[0,0,0,0,0,0]):
                $ 795 "direction(p[0,0,0,0,0,0],[0,1,0],8,120,160)"
                direction(p[0,0,0,0,0,0],[0,1,0],8,120,160)
                $ 796 "AAgcp≔get_actual_tcp_pose()"
                global AAgcp= get_actual_tcp_pose ()
                $ 797 "AAgangle≔up_right"
                global AAgangle=p[.445203173045, -.406687378356, -.031125942276, 2.308490741423, -1.066468937023, 1.322151316133]
                $ 798 "AAgtp≔p[AAgcp[0],AAgcp[1],AAgcp[2],AAgangle[3],AAgangle[4],AAgangle[5]]"
                global AAgtp=p[AAgcp[0],AAgcp[1],AAgcp[2],AAgangle[3],AAgangle[4],AAgangle[5]]
                $ 799 "MoveL"
                $ 800 "AAgtp" "breakAfter"
                movel(pose_trans(Base, AAgtp), a=0.08, v=0.08)
                $ 802 "for_z_VR1≔contact_fun(p[0,0,0,0,0,0],[0,0,-1],10000,15,15,  False)"
                global for_z_VR1=contact_fun(p[0,0,0,0,0,0],[0,0,-1],10000,15,15,  False)
                $ 803 "direction(p[0,0,0,0,0,0],[0,0,1],20,120,160)"
                direction(p[0,0,0,0,0,0],[0,0,1],20,120,160)
                $ 804 "write_welder(4, False )"
                write_welder(4,  False  )
              else:
                $ 805 "Else" "noBreak"
                $ 806 "for_z_VR1≔p[0,0,0,0,0,0]"
                global for_z_VR1=p[0,0,0,0,0,0]
              end
            end
          end
          $ 807 "HOR_MR"
          $ 808 "If A_Prepos_l[A_HOR_MR]≠p[0,0,0,0,0,0]"
          if (A_Prepos_l[A_HOR_MR] != p[0,0,0,0,0,0]):
            $ 809 "INIT"
            $ 810 "b2_left_par≔ False "
            global b2_left_par=  False
            $ 811 "b8_wv_2f≔ True "
            global b8_wv_2f=  True
            $ 812 "b7_tilt_degree≔[0,0,0]"
            global b7_tilt_degree=[0,0,0]
            $ 813 "A_sel_v≔A_HOR_MR"
            global A_sel_v=A_HOR_MR
            $ 814 "If b1_cell_info_R≟C or b1_cell_info_R≟D"
            if (b1_cell_info_R == C  or  b1_cell_info_R == D):
              $ 815 "wv_direction≔-1"
              global wv_direction=-1
              $ 816 "Call MoveFun_cd"
              MoveFun_cd()
              $ 817 "for_cal_xy≔contact_fun(p[0,0,0,0,0,0],[1,0,0],20000,20,20)"
              global for_cal_xy=contact_fun(p[0,0,0,0,0,0],[1,0,0],20000,20,20)
              $ 818 "direction(p[0,0,0,0,0,0],[-1,0,0],15,120,160)"
              direction(p[0,0,0,0,0,0],[-1,0,0],15,120,160)
              $ 819 "direction(p[0,0,0,0,0,0],[0,1,0],60,120,160)"
              direction(p[0,0,0,0,0,0],[0,1,0],60,120,160)
              $ 820 "direction(p[0,0,0,0,0,0],[1,0,0],20,120,160)"
              direction(p[0,0,0,0,0,0],[1,0,0],20,120,160)
              $ 821 "for_cal_x_wel≔contact_fun(p[0,0,0,0,0,0],[0,-1,0],20000,20,20)"
              global for_cal_x_wel=contact_fun(p[0,0,0,0,0,0],[0,-1,0],20000,20,20)
              $ 822 "direction(p[0,0,0,0,0,0],[0,1,0],20,120,160)"
              direction(p[0,0,0,0,0,0],[0,1,0],20,120,160)
              $ 823 "for_cal_y_wel≔contact_fun(p[0,0,0,0,0,0],[1,0,0],20000,20,20)"
              global for_cal_y_wel=contact_fun(p[0,0,0,0,0,0],[1,0,0],20000,20,20)
              $ 824 "direction(p[0,0,0,0,0,0],[-1,0,0],8,120,160)"
              direction(p[0,0,0,0,0,0],[-1,0,0],8,120,160)
              $ 825 "for_cal_zr≔contact_fun(p[0,0,0,0,0,0],[0,0,-1],20000,20,20)"
              global for_cal_zr=contact_fun(p[0,0,0,0,0,0],[0,0,-1],20000,20,20)
              $ 826 "direction(p[0,0,0,0,0,0],[0,0,1],20,120,160)"
              direction(p[0,0,0,0,0,0],[0,0,1],20,120,160)
              $ 827 "for_cal_rot≔A_Touch_p[A_HOR_R]"
              global for_cal_rot=A_Touch_p[A_HOR_R]
              $ 828 "A_Touch_p[A_sel_v]=p[for_cal_xy[0],for_cal_xy[1],for_cal_zr[2],for_cal_rot[3],for_cal_rot[4],for_cal_rot[5]]"
              A_Touch_p[A_sel_v]=p[for_cal_xy[0],for_cal_xy[1],for_cal_zr[2],for_cal_rot[3],for_cal_rot[4],for_cal_rot[5]]
              $ 829 "A_Touch_p[A_sel_v]=pose_trans(A_Touch_p[A_sel_v], p[-Touch_dis/1000,0,0,0,0,0])"
              A_Touch_p[A_sel_v]= pose_trans (A_Touch_p[A_sel_v], p[-Touch_dis/1000,0,0,0,0,0])
              $ 830 "write_welder(4, False )"
              write_welder(4,  False  )
            else:
              $ 831 "Else" "noBreak"
              $ 832 "wv_direction≔-1"
              global wv_direction=-1
              $ 833 "for_cal_rot≔A_Touch_p[A_HOR_R]"
              global for_cal_rot=A_Touch_p[A_HOR_R]
              $ 834 "Call MoveFun_cd"
              MoveFun_cd()
              $ 835 "for_cal_y_wel≔contact_fun(p[0,0,0,0,0,0],[1,0,0],20000,20,20)"
              global for_cal_y_wel=contact_fun(p[0,0,0,0,0,0],[1,0,0],20000,20,20)
              $ 836 "vr2_p1≔for_cal_y_wel"
              global vr2_p1=for_cal_y_wel
              $ 837 "for_cal_y_wel[2]=for_cal_rot[2]"
              for_cal_y_wel[2]=for_cal_rot[2]
              $ 838 "dir_x_cal≔get_feature_Line(for_cal_rot,for_cal_y_wel)"
              global dir_x_cal=get_feature_Line(for_cal_rot,for_cal_y_wel)
              $ 839 "vr2_p2≔feature_offset(vr2_p1,p[0,0.02,0,0,0,0],dir_x_cal)"
              global vr2_p2=feature_offset(vr2_p1,p[0,0.02,0,0,0,0],dir_x_cal)
              $ 840 "direction(p[0,0,0,0,0,0],[-1,0,0],40,120,160)"
              direction(p[0,0,0,0,0,0],[-1,0,0],40,120,160)
              $ 841 "direction(p[0,0,0,0,0,0],[0,1,0],80,120,160)"
              direction(p[0,0,0,0,0,0],[0,1,0],80,120,160)
              $ 842 "for_cal_y_wel≔contact_fun(p[0,0,0,0,0,0],[1,0,0],20000,20,20)"
              global for_cal_y_wel=contact_fun(p[0,0,0,0,0,0],[1,0,0],20000,20,20)
              $ 843 "direction(p[0,0,0,0,0,0],[-1,0,0],5,120,160)"
              direction(p[0,0,0,0,0,0],[-1,0,0],5,120,160)
              $ 844 "direction(p[0,0,0,0,0,0],[0,-1,0],60,120,160)"
              direction(p[0,0,0,0,0,0],[0,-1,0],60,120,160)
              $ 845 "direction(p[0,0,0,0,0,0],[1,0,0],7,120,160)"
              direction(p[0,0,0,0,0,0],[1,0,0],7,120,160)
              $ 846 "for_cal_x_wel≔contact_fun(p[0,0,0,0,0,0],[0,1,0],20000,20,20)"
              global for_cal_x_wel=contact_fun(p[0,0,0,0,0,0],[0,1,0],20000,20,20)
              $ 847 "vr2_p3≔for_cal_x_wel"
              global vr2_p3=for_cal_x_wel
              $ 848 "get_ml≔get_feature_pose(for_cal_x_wel,for_cal_rot)"
              global get_ml=get_feature_pose(for_cal_x_wel,for_cal_rot)
              $ 850 "A_Touch_p[A_sel_v]=feature_offset(for_cal_rot,p[0,-get_ml[0]+(-cd_offset+cd_extra_dis)/1000,0,0,0,0],dir_x_cal)"
              A_Touch_p[A_sel_v]=feature_offset(for_cal_rot,p[0,-get_ml[0]+(-cd_offset+cd_extra_dis)/1000,0,0,0,0],dir_x_cal)
              $ 851 "vr2_p4≔A_Touch_p[A_HOR_MR]"
              global vr2_p4=A_Touch_p[A_HOR_MR]
              $ 852 "direction(p[0,0,0,0,0,0],[0,-1,0],5,120,160)"
              direction(p[0,0,0,0,0,0],[0,-1,0],5,120,160)
              $ 853 "direction(p[0,0,0,0,0,0],[-1,0,0],20,120,160)"
              direction(p[0,0,0,0,0,0],[-1,0,0],20,120,160)
              $ 854 "write_welder(4, False )"
              write_welder(4,  False  )
            end
            $ 855 "homeing()"
            homeing()
            $ 856 "wv_direction≔1"
            global wv_direction=1
          else:
            $ 857 "Else" "noBreak"
            $ 858 "homeing()"
            homeing()
          end
          $ 859 "VR2"
          $ 860 "If A_Prepos_l[A_VR2]≠p[0,0,0,0,0,0]"
          if (A_Prepos_l[A_VR2] != p[0,0,0,0,0,0]):
            $ 861 "Init"
            $ 862 "b2_left_par≔ False "
            global b2_left_par=  False
            $ 863 "b8_wv_2f≔ False "
            global b8_wv_2f=  False
            $ 864 "b7_tilt_degree≔basic_tilt_3f"
            global b7_tilt_degree=basic_tilt_3f
            $ 865 "A_sel_v≔A_VR2"
            global A_sel_v=A_VR2
            $ 866 "A_sel_v_end≔A_VR2_END"
            global A_sel_v_end=A_VR2_END
            $ 867 "b2_par_cd≔1"
            global b2_par_cd=1
            $ 868 "If b1_cell_info_R≟A or b1_cell_info_R≟C or b1_cell_info_R≟c"
            if (b1_cell_info_R == A  or  b1_cell_info_R == C  or  b1_cell_info_R == c):
              $ 869 "Scallup_check≔ True "
              global Scallup_check=  True
            else:
              $ 870 "Else" "noBreak"
              $ 871 "Scallup_check≔ False "
              global Scallup_check=  False
            end
            $ 872 "If b1_cell_info_R≟d or b1_cell_info_R≟c"
            if (b1_cell_info_R == d  or  b1_cell_info_R == c):
              $ 873 "Halt"
              halt
              $ 874 "If vr2_p1≟p[0,0,0,0,0,0]"
              if (vr2_p1 == p[0,0,0,0,0,0]):
                $ 875 "Call MoveFun_cd"
                MoveFun_cd()
                $ 876 "vr2_p1≔contact_fun(p[0,0,0,0,0,0],[1,0,0],20000,20,20)"
                global vr2_p1=contact_fun(p[0,0,0,0,0,0],[1,0,0],20000,20,20)
                $ 877 "direction(p[0,0,0,0,0,0],[-1,0,0],20,120,160)"
                direction(p[0,0,0,0,0,0],[-1,0,0],20,120,160)
                $ 878 "direction(p[0,0,0,0,0,0],[0,1,0],10,120,160)"
                direction(p[0,0,0,0,0,0],[0,1,0],10,120,160)
                $ 879 "vr2_p2≔contact_fun(p[0,0,0,0,0,0],[1,0,0],20000,20,20)"
                global vr2_p2=contact_fun(p[0,0,0,0,0,0],[1,0,0],20000,20,20)
                $ 880 "direction(p[0,0,0,0,0,0],[-1,0,0],14,120,160)"
                direction(p[0,0,0,0,0,0],[-1,0,0],14,120,160)
                $ 881 "vr2_p3≔contact_fun(p[0,0,0,0,0,0],[0,1,0],20000,20,20)"
                global vr2_p3=contact_fun(p[0,0,0,0,0,0],[0,1,0],20000,20,20)
                $ 882 "direction(p[0,0,0,0,0,0],[0,-1,0],30,120,160)"
                direction(p[0,0,0,0,0,0],[0,-1,0],30,120,160)
                $ 883 "direction(p[0,0,0,0,0,0],[-1,0,0],20,120,160)"
                direction(p[0,0,0,0,0,0],[-1,0,0],20,120,160)
                $ 884 "vr2_p4≔contact_fun(p[0,0,0,0,0,0],[0,0,-1],20000,20,20)"
                global vr2_p4=contact_fun(p[0,0,0,0,0,0],[0,0,-1],20000,20,20)
                $ 885 "direction(p[0,0,0,0,0,0],[0,0,1],40,120,160)"
                direction(p[0,0,0,0,0,0],[0,0,1],40,120,160)
                $ 886 "A_Touch_p[A_sel_v]=touch_xyz_get_middle(vr2_p1,vr2_p2,vr2_p3,vr2_p4)"
                A_Touch_p[A_sel_v]=touch_xyz_get_middle(vr2_p1,vr2_p2,vr2_p3,vr2_p4)
                $ 887 "var_4≔A_Touch_p[A_sel_v]"
                global var_4=A_Touch_p[A_sel_v]
                $ 888 "var_4≔pose_trans(var_4, p[a6_callar_vert/1000,0,0,0,0,0])"
                global var_4= pose_trans (var_4, p[a6_callar_vert/1000,0,0,0,0,0])
                $ 889 "var_5≔get_actual_tcp_pose()"
                global var_5= get_actual_tcp_pose ()
                $ 890 "var_5[2]=var_4[2]"
                var_5[2]=var_4[2]
                $ 891 "var_5≔pose_trans(var_5, p[0,0,0,0,d2r(10),0])"
                global var_5= pose_trans (var_5, p[0,0,0,0,d2r(10),0])
                $ 892 "MoveL"
                $ 893 "var_5" "breakAfter"
                movel(pose_trans(Base, var_5), a=0.1, v=0.1)
                $ 894 "vr2_p1_up≔contact_fun(p[0,0,0,0,0,0],[1,0,0],20000,20,20)"
                global vr2_p1_up=contact_fun(p[0,0,0,0,0,0],[1,0,0],20000,20,20)
                $ 895 "direction(p[0,0,0,0,0,0],[-1,0,0],20,120,160)"
                direction(p[0,0,0,0,0,0],[-1,0,0],20,120,160)
                $ 896 "direction(p[0,0,0,0,0,0],[0,1,0],10,120,160)"
                direction(p[0,0,0,0,0,0],[0,1,0],10,120,160)
                $ 897 "vr2_p2_up≔contact_fun(p[0,0,0,0,0,0],[1,0,0],20000,20,20)"
                global vr2_p2_up=contact_fun(p[0,0,0,0,0,0],[1,0,0],20000,20,20)
                $ 898 "direction(p[0,0,0,0,0,0],[-1,0,0],14,120,160)"
                direction(p[0,0,0,0,0,0],[-1,0,0],14,120,160)
